# B&R Automation Studio project MotionTestBenchMaster (part 8)

#### SIKO_FB.st - Siko Manager
```iecst
(********************************************************************
 * COPYRIGHT - Sidel SpA
 ********************************************************************
 * Library: SIDEL
 * File: SIKO_FB.st
 * Author: 100383
 * Created: November 16, 2015
 ********************************************************************
 * Implementation of library SIDEL_CNTR
 ********************************************************************)

FUNCTION_BLOCK Siko_FB

	memset(ADR(Com),0,SIZEOF(Com));

	DeviceData.EmergencyOkFbk := IN_EmergencyOK;

	IF NOT IN_CommunicationOK THEN
		DeviceData.PositioningInProgress := FALSE;
		DeviceData.InPosition := FALSE;
		CounterRead := 0;
		CounterWrite := 0;
		DeviceData.CalibrationInProgress := FALSE;
		DeviceData.CommunicationFault := TRUE;
		RETURN;
	ELSE
		DeviceData.CommunicationFault := FALSE;
	END_IF

	IF CounterRead <> 0 OR CounterWrite <> 0 OR (DeviceData.CalibrationInProgress AND NOT DeviceData.Calibrate) THEN
		DeviceData.ReadOrWriteInProgress := TRUE;
	ELSE
		DeviceData.ReadOrWriteInProgress := FALSE;
	END_IF

	TReadAndWrite(IN:= DeviceData.ReadOrWriteInProgress, PT:= t#30s);
	DeviceData.ReadOrWriteError := TReadAndWrite.Q;

	IF DeviceData.ReadOrWriteError OR IN_Reset THEN
		CounterRead := 0;
		CounterWrite := 0;
		DeviceData.CalibrationInProgress := FALSE;
	END_IF

	Com.SIKO_FLR	:= IO.SIKO_FLR;
	Temp_HIW		:= IO.SIKO_FLR.HIW_L + (IO.SIKO_FLR.HIW_H * 16#10000);
	Temp_IN_PWE		:= IO.SIKO_FLR.PWE_L + (IO.SIKO_FLR.PWE_H * 16#10000);

	IF DeviceData.Data.SpindlePitch = 0 THEN
		KFactorReal := 1.0;
	ELSE
		KFactorReal := 100.0;
	END_IF

	DeviceData.CurrentPos := UDINT_TO_REAL(Temp_HIW) / KFactorReal;

	DeviceData.TargetOutsideSwLimit := (DeviceData.TargetPos > DeviceData.Data.UpperLimit) OR (DeviceData.TargetPos < DeviceData.Data.LowerLimit);

	IF EDGEPOS(DeviceData.StartPositioning AND IN_EmergencyOK AND NOT DeviceData.MotorDisabled AND NOT DeviceData.TargetOutsideSwLimit) THEN
		DeviceData.PositioningInProgress := TRUE;
	END_IF

	DeviceData.InPosition := ABS(DeviceData.TargetPos - DeviceData.CurrentPos) <= DeviceData.Data.PosWindows;

	SwitchOn := DeviceData.JogBackward OR DeviceData.JogForward OR DeviceData.PositioningInProgress;

	TPowerOn(IN:= SwitchOn, PT:= t#20s);

	Com.FLR_SIKO.STW.0 := IN_EmergencyOK AND TPowerOn.Q AND DeviceData.Enable AND NOT DeviceData.OnError;
	Com.FLR_SIKO.STW.1 := IN_EmergencyOK AND TPowerOn.Q AND DeviceData.Enable AND NOT DeviceData.OnError;

	Com.FLR_SIKO.STW.7 := IN_Reset;

	Com.FLR_SIKO.STW.5 := Com.SIKO_FLR.ZSW.2 AND NOT DeviceData.AbortPositioning;
	Com.FLR_SIKO.STW.4 := Com.SIKO_FLR.ZSW.2 AND NOT DeviceData.AbortPositioning;

	Com.FLR_SIKO.STW.3 := Com.SIKO_FLR.ZSW.4;

	IF DeviceData.Enable THEN
		DeviceData.MotorDisabled := FALSE;
	ELSIF NOT DeviceData.Enable AND NOT Com.SIKO_FLR.ZSW.4 THEN
		DeviceData.MotorDisabled := TRUE;
	END_IF

	DeviceData.OnError := Com.SIKO_FLR.ZSW.3;

	DeviceData.Warning := Com.SIKO_FLR.ZSW.8 AND Com.SIKO_FLR.ZSW.7;

	DeviceData.DeviceOutsideSwLimit := Com.SIKO_FLR.ZSW.14 OR (DeviceData.CurrentPos > DeviceData.Data.UpperLimit) OR (DeviceData.CurrentPos < DeviceData.Data.LowerLimit);

	Com.FLR_SIKO.STW.9 := Com.SIKO_FLR.ZSW.2 AND NOT DeviceData.OnError AND NOT DeviceData.PositioningInProgress AND	(DeviceData.JogForward XOR DeviceData.JogBackward);

	Com.FLR_SIKO.STW.15 := Com.FLR_SIKO.STW.9 AND DeviceData.JogBackward;

	Com.FLR_SIKO.STW.6 := DeviceData.PositioningInProgress AND NOT DeviceData.OnError AND Com.SIKO_FLR.ZSW.15 AND Com.SIKO_FLR.ZSW.13;

	IF Com.FLR_SIKO.STW.6 THEN
		Temp_HSW := REAL_TO_UDINT(DeviceData.TargetPos * KFactorReal);
	END_IF

	PositionFinished := ABS(DeviceData.TargetPos - DeviceData.CurrentPos) <= DeviceData.Data.PosWindows;

	IF DeviceData.TargetOutsideSwLimit OR DeviceData.OnError OR NOT IN_EmergencyOK OR DeviceData.MotorDisabled OR
	(DeviceData.InPosition AND Com.SIKO_FLR.ZSW.13) OR
	(PositionFinished AND Com.SIKO_FLR.ZSW.13) OR
	EDGEPOS(DeviceData.AbortPositioning) THEN
		DeviceData.PositioningInProgress := FALSE;
	END_IF

	RisingFrontRead := EDGEPOS((DeviceData.StartRead AND NOT DeviceData.ReadOrWriteInProgress) OR ReloadData);

	Com.FLR_SIKO.PKE := 0;

	IF NOT DeviceData.ReadOrWriteError THEN
		IF RisingFrontRead THEN
			CounterRead := 1;
			ReloadData := FALSE;
		END_IF

		CASE CounterRead OF
			1:	// Operative Mode
				Com.FLR_SIKO.PKE := 16#13A2;

				IF Com.SIKO_FLR.PKE = 16#13A2 THEN
					DeviceData.Data.OperationMode := UDINT_TO_INT(Temp_IN_PWE);
					CounterRead := CounterRead  + 1;
				END_IF

			2:	// Error Buffer [0]
				Com.FLR_SIKO.IND := 0;
				Com.FLR_SIKO.PKE := 16#63B1;

				IF Com.SIKO_FLR.PKE = 16#43B1 THEN
					IF Com.SIKO_FLR.IND = 0 THEN
						DeviceData.Data.FaultBuffer0 := UDINT_TO_INT(Temp_IN_PWE);
						CounterRead := CounterRead  + 1;
					END_IF
				END_IF

			3:	// Error Buffer [1]
				Com.FLR_SIKO.IND := 1;
				Com.FLR_SIKO.PKE := 16#63B1;

				IF Com.SIKO_FLR.PKE = 16#43B1 THEN
					IF Com.SIKO_FLR.IND = 1 THEN
						DeviceData.Data.FaultBuffer1 := UDINT_TO_INT(Temp_IN_PWE);
						CounterRead := CounterRead  + 1;
					END_IF
				END_IF

			4:	// Error Buffer [2]
				Com.FLR_SIKO.IND := 2;
				Com.FLR_SIKO.PKE := 16#63B1;

				IF Com.SIKO_FLR.PKE = 16#43B1 THEN
					IF Com.SIKO_FLR.IND = 2 THEN
						DeviceData.Data.FaultBuffer2 := UDINT_TO_INT(Temp_IN_PWE);
						CounterRead := CounterRead  + 1;
					END_IF
				END_IF

			5:	// Error Buffer [3]
				Com.FLR_SIKO.IND := 3;
				Com.FLR_SIKO.PKE := 16#63B1;

				IF Com.SIKO_FLR.PKE = 16#43B1 THEN
					IF Com.SIKO_FLR.IND = 3 THEN
						DeviceData.Data.FaultBuffer3 := UDINT_TO_INT(Temp_IN_PWE);
						CounterRead := CounterRead  + 1;
					END_IF
				END_IF

			6:	// Error Buffer [4]
				Com.FLR_SIKO.IND := 4;
				Com.FLR_SIKO.PKE := 16#63B1;

				IF Com.SIKO_FLR.PKE = 16#43B1 THEN
					IF Com.SIKO_FLR.IND = 4 THEN
						DeviceData.Data.FaultBuffer4 := UDINT_TO_INT(Temp_IN_PWE);
						CounterRead := CounterRead  + 1;
					END_IF
				END_IF

			7:	// Error Buffer [5]
				Com.FLR_SIKO.IND := 5;
				Com.FLR_SIKO.PKE := 16#63B1;

				IF Com.SIKO_FLR.PKE = 16#43B1 THEN
					IF Com.SIKO_FLR.IND = 5 THEN
						DeviceData.Data.FaultBuffer5 := UDINT_TO_INT(Temp_IN_PWE);
						CounterRead := CounterRead  + 1;
					END_IF
				END_IF

			8:	// Error Buffer [6]
				Com.FLR_SIKO.IND := 6;
				Com.FLR_SIKO.PKE := 16#63B1;

				IF Com.SIKO_FLR.PKE = 16#43B1 THEN
					IF Com.SIKO_FLR.IND = 6 THEN
						DeviceData.Data.FaultBuffer6 := UDINT_TO_INT(Temp_IN_PWE);
						CounterRead := CounterRead  + 1;
					END_IF
				END_IF

			9:	// Error Buffer [7]
				Com.FLR_SIKO.IND := 7;
				Com.FLR_SIKO.PKE := 16#63B1;

				IF Com.SIKO_FLR.PKE = 16#43B1 THEN
					IF Com.SIKO_FLR.IND = 7 THEN
						DeviceData.Data.FaultBuffer7 := UDINT_TO_INT(Temp_IN_PWE);
						CounterRead := CounterRead  + 1;
					END_IF
				END_IF

			10:	// Error Buffer [8]
				Com.FLR_SIKO.IND := 8;
				Com.FLR_SIKO.PKE := 16#63B1;

				IF Com.SIKO_FLR.PKE = 16#43B1 THEN
					IF Com.SIKO_FLR.IND = 8 THEN
						DeviceData.Data.FaultBuffer8 := UDINT_TO_INT(Temp_IN_PWE);
						CounterRead := CounterRead  + 1;
					END_IF
				END_IF

			11:	// Error Buffer [9]
				Com.FLR_SIKO.IND := 9;
				Com.FLR_SIKO.PKE := 16#63B1;

				IF Com.SIKO_FLR.PKE = 16#43B1 THEN
					IF Com.SIKO_FLR.IND = 9 THEN
						DeviceData.Data.FaultBuffer9 := UDINT_TO_INT(Temp_IN_PWE);
						CounterRead := CounterRead  + 1;
					END_IF
				END_IF

			12:	// P Gain
				Com.FLR_SIKO.PKE := 16#13E8;

				IF Com.SIKO_FLR.PKE = 16#13E8 THEN
					DeviceData.Data.PGain := UDINT_TO_INT(Temp_IN_PWE);
					CounterRead := CounterRead  + 1;
				END_IF

			13:	// I Gain
				Com.FLR_SIKO.PKE := 16#13E9;

				IF Com.SIKO_FLR.PKE = 16#13E9 THEN
					DeviceData.Data.IGain := UDINT_TO_INT(Temp_IN_PWE);
					CounterRead := CounterRead  + 1;
				END_IF

			14:	// D Gain
				Com.FLR_SIKO.PKE := 16#13EA;

				IF Com.SIKO_FLR.PKE = 16#13EA THEN
					DeviceData.Data.DGain := UDINT_TO_INT(Temp_IN_PWE);
					CounterRead := CounterRead  + 1;
				END_IF

			15:	// A Pos
				Com.FLR_SIKO.PKE := 16#13EB;

				IF Com.SIKO_FLR.PKE = 16#13EB THEN
					DeviceData.Data.APos := UDINT_TO_INT(Temp_IN_PWE);
					CounterRead := CounterRead  + 1;
				END_IF

			16:	// V Pos
				Com.FLR_SIKO.PKE := 16#13EC;

				IF Com.SIKO_FLR.PKE = 16#13EC THEN
					DeviceData.Data.VPos := UDINT_TO_INT(Temp_IN_PWE);
					CounterRead := CounterRead  + 1;
				END_IF

			17:	// V Jog
				Com.FLR_SIKO.PKE := 16#13F0;

				IF Com.SIKO_FLR.PKE = 16#13F0 THEN
					DeviceData.Data.VJog := UDINT_TO_INT(Temp_IN_PWE);
					CounterRead := CounterRead  + 1;
				END_IF

			18:	// SpindlePitch
				Com.FLR_SIKO.PKE := 16#13F4;

				IF Com.SIKO_FLR.PKE = 16#13F4 THEN
					DeviceData.Data.SpindlePitch := UDINT_TO_INT(Temp_IN_PWE) / 100;
					CounterRead := CounterRead  + 1;
				END_IF

			19:	// GearIn
				Com.FLR_SIKO.PKE := 16#13F2;

				IF Com.SIKO_FLR.PKE = 16#13F2 THEN
					DeviceData.Data.GearIn := UDINT_TO_INT(Temp_IN_PWE);
					CounterRead := CounterRead  + 1;
				END_IF

			20:	// GearOut
				Com.FLR_SIKO.PKE := 16#13F3;

				IF Com.SIKO_FLR.PKE = 16#13F3 THEN
					DeviceData.Data.GearOut := UDINT_TO_INT(Temp_IN_PWE);
					CounterRead := CounterRead  + 1;
				END_IF

			21:	// Toll Pos
				Com.FLR_SIKO.PKE := 16#13F1;

				IF Com.SIKO_FLR.PKE = 16#13F1 THEN
					DeviceData.Data.PosWindows := UDINT_TO_REAL(Temp_IN_PWE) / KFactorReal;
					CounterRead := CounterRead  + 1;
				END_IF

			22:	// Rotation
				Com.FLR_SIKO.PKE := 16#13F5;

				IF Com.SIKO_FLR.PKE = 16#13F5 THEN
					DeviceData.Data.SenseOfRotation := UDINT_TO_INT(Temp_IN_PWE);
					CounterRead := CounterRead  + 1;
				END_IF

			23:	// Upper limit
				Com.FLR_SIKO.PKE := 16#13F8;

				IF Com.SIKO_FLR.PKE = 16#13F8 OR Com.SIKO_FLR.PKE = 16#23F8 THEN
					DeviceData.Data.UpperLimit := UDINT_TO_REAL(Temp_IN_PWE) / KFactorReal;
					CounterRead := CounterRead  + 1;
				END_IF

			24:	// Lower limit
				Com.FLR_SIKO.PKE := 16#13F9;

				IF Com.SIKO_FLR.PKE = 16#13F9 OR Com.SIKO_FLR.PKE = 16#23F9 THEN
					DeviceData.Data.LowerLimit := UDINT_TO_REAL(Temp_IN_PWE) / KFactorReal;
					CounterRead := CounterRead  + 1;
				END_IF

			25:	// Calibration value
				Com.FLR_SIKO.PKE := 16#13FA;

				IF Com.SIKO_FLR.PKE = 16#13FA OR Com.SIKO_FLR.PKE = 16#23FA THEN
					DeviceData.Data.CalibrationValue := UDINT_TO_REAL(Temp_IN_PWE) / KFactorReal;
					CounterRead := CounterRead  + 1;
				END_IF

			26:	// Status word
				Com.FLR_SIKO.PKE := 16#13FC;

				IF Com.SIKO_FLR.PKE = 16#13FC THEN
					DeviceData.Data.SystemStatusWord := UDINT_TO_INT(Temp_IN_PWE);
					CounterRead := 0;
				END_IF

		END_CASE
	END_IF

	DeviceData.WriteEnabled := (DeviceData.MotorDisabled OR NOT DeviceData.PositioningInProgress) AND NOT DeviceData.ReadOrWriteInProgress AND NOT DeviceData.ReadOrWriteError AND NOT DeviceData.IllegalOperation;

	RisingFrontWrite := EDGEPOS(DeviceData.StartWrite);

	IF RisingFrontWrite AND DeviceData.WriteEnabled AND NOT DeviceData.ReadOrWriteError THEN
		DeviceData.Data.TimeoutPositioning	:= IN_TimeOutPositioning;
		DeviceData.Data.PosWindows			:= IN_PosWindows;
		DeviceData.Data.UpperLimit			:= IN_UpperLimit;
		DeviceData.Data.LowerLimit			:= IN_LowerLimit;
		DeviceData.Data.CalibrationValue	:= IN_CalibrationValue;

		DeviceData.Data.PGain			:= REAL_TO_INT(IN_PGain);
		DeviceData.Data.IGain			:= REAL_TO_INT(IN_IGain);
		DeviceData.Data.DGain			:= REAL_TO_INT(IN_DGain);
		DeviceData.Data.VPos			:= REAL_TO_INT(IN_VPos);
		DeviceData.Data.APos			:= REAL_TO_INT(IN_APos);
		DeviceData.Data.VJog			:= REAL_TO_INT(IN_VJog);
		DeviceData.Data.GearIn			:= REAL_TO_INT(IN_GearIn);
		DeviceData.Data.GearOut			:= REAL_TO_INT(IN_GearOut);
		DeviceData.Data.SpindlePitch	:= REAL_TO_INT(IN_SpindlePitch);
		DeviceData.Data.SenseOfRotation	:= REAL_TO_INT(IN_SenseOfRotation);
	END_IF

	IF NOT DeviceData.ReadOrWriteError THEN
		IF RisingFrontWrite THEN
			CounterWrite := 1;
		END_IF

		CASE CounterWrite OF
			1:	// Op Mode
				Com.FLR_SIKO.PKE := 16#23A2;
				Temp_OUT_PWE := 2;

				IF Com.SIKO_FLR.PKE = 16#13A2 THEN
					CounterWrite := CounterWrite + 1;
				END_IF

			2:	// Proportional Gain
				Com.FLR_SIKO.PKE := 16#23E8;
				Temp_OUT_PWE := DeviceData.Data.PGain;

				IF Com.SIKO_FLR.PKE = 16#13E8 THEN
					CounterWrite := CounterWrite + 1;
				END_IF

			3:	// Integral Gain
				Com.FLR_SIKO.PKE := 16#23E9;
				Temp_OUT_PWE := DeviceData.Data.IGain;

				IF Com.SIKO_FLR.PKE = 16#13E9 THEN
					CounterWrite := CounterWrite + 1;
				END_IF

			4:	// Derivative Gain
				Com.FLR_SIKO.PKE := 16#23EA;
				Temp_OUT_PWE := DeviceData.Data.DGain;

				IF Com.SIKO_FLR.PKE = 16#13EA THEN
					CounterWrite := CounterWrite + 1;
				END_IF

			5:	// Acc Positioning
				Com.FLR_SIKO.PKE := 16#23EB;
				Temp_OUT_PWE := DeviceData.Data.APos;

				IF Com.SIKO_FLR.PKE = 16#13EB THEN
					CounterWrite := CounterWrite + 1;
				END_IF

			6:	// Speed Positioning
				Com.FLR_SIKO.PKE := 16#23EC;
				Temp_OUT_PWE := DeviceData.Data.VPos;

				IF Com.SIKO_FLR.PKE = 16#13EC THEN
					CounterWrite := CounterWrite + 1;
				END_IF

			7:	// Speed Jog
				Com.FLR_SIKO.PKE := 16#23F0;
				Temp_OUT_PWE := DeviceData.Data.VJog;

				IF Com.SIKO_FLR.PKE = 16#13F0 THEN
					CounterWrite := CounterWrite + 1;
				END_IF

			8:	// GearIn
				Com.FLR_SIKO.PKE := 16#23F2;
				Temp_OUT_PWE := DeviceData.Data.GearIn;

				IF Com.SIKO_FLR.PKE = 16#13F2 THEN
					CounterWrite := CounterWrite + 1;
				END_IF

			9:	// GearOut
				Com.FLR_SIKO.PKE := 16#23F3;
				Temp_OUT_PWE := DeviceData.Data.GearOut;

				IF Com.SIKO_FLR.PKE = 16#13F3 THEN
					CounterWrite := CounterWrite + 1;
				END_IF

			10:	// SpinlePitch
				Com.FLR_SIKO.PKE := 16#23F4;
				Temp_OUT_PWE := DeviceData.Data.SpindlePitch * 100 ;

				IF Com.SIKO_FLR.PKE = 16#13F4 THEN
					CounterWrite := CounterWrite + 1;
				END_IF

			11:	// Position Windows
				Com.FLR_SIKO.PKE := 16#23F1;
				Temp_OUT_PWE := REAL_TO_INT(DeviceData.Data.PosWindows * KFactorReal);

				IF Com.SIKO_FLR.PKE = 16#13F1 THEN
					CounterWrite := CounterWrite + 1;
				END_IF

			12:	// Rotatation
				Com.FLR_SIKO.PKE := 16#23F5;
				Temp_OUT_PWE := DeviceData.Data.SenseOfRotation;

				IF Com.SIKO_FLR.PKE = 16#13F5 THEN
					CounterWrite := CounterWrite + 1;
				END_IF

			13:	// Upper Limit
				Com.FLR_SIKO.PKE := 16#33F8;
				Temp_OUT_PWE := REAL_TO_UDINT(DeviceData.Data.UpperLimit * KFactorReal);

				IF Com.SIKO_FLR.PKE = 16#23F8 THEN
					CounterWrite := CounterWrite + 1;
				ELSIF Com.SIKO_FLR.PKE = 16#73F8 THEN
					CounterWrite := CounterWrite + 2;
				END_IF

			14:	// Lower Limit
				Com.FLR_SIKO.PKE := 16#33F9;
				Temp_OUT_PWE := REAL_TO_UDINT(DeviceData.Data.LowerLimit * KFactorReal);

				IF Com.SIKO_FLR.PKE = 16#23F9 THEN
					CounterWrite := 50;
				END_IF

			15:	//Upper Limit error - Write Lower Limit
				Com.FLR_SIKO.PKE := 16#33F9;
				Temp_OUT_PWE := REAL_TO_UDINT(DeviceData.Data.LowerLimit * KFactorReal);

				IF Com.SIKO_FLR.PKE = 16#23F9 THEN
					CounterWrite := CounterWrite + 1;
				END_IF

			16: //Upper Limit error - Reweite Upper limit
				Com.FLR_SIKO.PKE := 16#33F8;
				Temp_OUT_PWE := REAL_TO_UDINT(DeviceData.Data.UpperLimit * KFactorReal);

				IF Com.SIKO_FLR.PKE = 16#23F8 THEN
					CounterWrite	:= 50;
				END_IF

			50: //Reset PWE
				Temp_OUT_PWE	:= 0;
				CounterWrite	:= 0;
				ReloadData := TRUE;
		END_CASE
	END_IF

	IF EDGEPOS(DeviceData.Calibrate AND DeviceData.WriteEnabled) THEN
		CounterCalibration := 1;
	END_IF

	CASE CounterCalibration OF
		1:
			DeviceData.Data.CalibrationValue := IN_CalibrationValue;
			DeviceData.CalibrationDone := FALSE;
			CounterCalibration := CounterCalibration + 1;

		2://Write Calibration Data
			Com.FLR_SIKO.PKE := 16#33FA;
			Temp_OUT_PWE := REAL_TO_UDINT(DeviceData.Data.CalibrationValue * KFactorReal);
			DeviceData.CalibrationInProgress := TRUE;

			IF Com.SIKO_FLR.PKE = 16#23FA THEN
				CounterCalibration := CounterCalibration + 1;
			END_IF

		3://Check Calibration Data
			IF ABS(Temp_IN_PWE - Temp_HIW) < 5 THEN
				DeviceData.CalibrationDone := TRUE;
				DeviceData.CalibrationInProgress := FALSE;
				CounterCalibration := 0;
			END_IF
	END_CASE

	IF ((DeviceData.Calibrate AND NOT DeviceData.CalibrationInProgress) OR RisingFrontWrite) AND NOT DeviceData.WriteEnabled THEN
		DeviceData.IllegalOperation := TRUE;
	ELSIF DeviceData.IllegalOperation AND IN_Reset THEN
		DeviceData.IllegalOperation := FALSE;
	END_IF

	IO.FLR_SIKO := Com.FLR_SIKO;
	IO.FLR_SIKO.PWE_H := UDINT_TO_UINT(SHR(Temp_OUT_PWE, 16));
	IO.FLR_SIKO.PWE_L := UDINT_TO_UINT(Temp_OUT_PWE AND 16#FFFF);
	IO.FLR_SIKO.HSW_H := UDINT_TO_UINT(SHR(Temp_HSW, 16));
	IO.FLR_SIKO.HSW_L := UDINT_TO_UINT(Temp_HSW AND 16#FFFF) ;

END_FUNCTION_BLOCK
```

#### PID_FF_Mod.st - FF calculation
```iecst
FUNCTION_BLOCK PID_FF_Mod
	IF SP1_ON THEN
		FF_SP2_Save := IN_FF_SP2;
		IF FF_SP2_Save >= IN_FF_SP1 THEN
			FF_SP2_Save := IN_FF_SP1;
		END_IF
		FF_SP2_Time.PT := REAL_TO_TIME(IN_SP1_SP2_Time/1000);
	END_IF

	FF_SP2_Time.IN := SP1_ON;
	FF_SP2_Time();

	IF NOT IN_Reset AND IN_Enable THEN
		IF ( IN_Raise_Step_Counter >= IN_Raise_Step ) OR ( IN_Raise_Step_Counter >= 100 ) THEN
			Running := TRUE;
			Lower_Ramp := TRUE;
		END_IF
	END_IF

	IF (NOT IN_Enable AND (( IN_Lower_Step_Counter >= IN_Lower_Step ) OR ( IN_Lower_Step_Counter >= 100 )))
		OR IN_Reset THEN
		Running := FALSE;
		SP1_ON := FALSE;
		SP2_ON := FALSE;
	END_IF

	FF_SP1_Recipe := (IN_FF_SP1);
	FF_SP2_Recipe := (IN_FF_SP2);
	Speed := IN_Actual_Speed;
	Max_Speed := MAX(IN_Size_Speed, 1);

	FF_SP1_Val := FF_SP1_Recipe * Speed;
	FF_SP1_Val := FF_SP1_Val / Max_Speed;

	FF_SP2_Val := FF_SP2_Recipe * Speed;
	FF_SP2_Val := FF_SP2_Val / Max_Speed;

	IF NOT Running AND NOT Lower_Ramp THEN
		FF_value_Out := 0.0;
	ELSIF NOT Running THEN
		Ramp_Time := 200.0;
		Ramp_Speed_R := (IN_Ramp_Speed);
		Ramp_Value := Ramp_Value - ((Ramp_Time /1000.0) * Ramp_Speed_R );
		IF Ramp_Value <= 0 THEN
			Lower_Ramp := FALSE;
			Ramp_Value := 0;
		END_IF
		FF_value_Out := Ramp_Value;
	ELSIF SP2_ON THEN
		FF_value_Out := FF_SP2_Val;
		Ramp_Value := FF_SP2_Val;
	ELSIF FF_SP2_Time.Q THEN
		Ramp_Time := 200.0;
		Ramp_Speed_R := (IN_Ramp_Speed);
		Ramp_Value := Ramp_Value - ((Ramp_Time /1000.0) * Ramp_Speed_R );
		IF Ramp_Value <= FF_SP2_Val THEN
			SP2_ON := TRUE;
			Ramp_Value := FF_SP2_Val;
		END_IF
		FF_value_Out := Ramp_Value;
	ELSIF SP1_ON THEN
		FF_value_Out := FF_SP1_Val;
		Ramp_Value := FF_SP1_Val;
	ELSE
		Ramp_Time := 200.0;
		Ramp_Speed_R := (IN_Ramp_Speed);
		Ramp_Value := Ramp_Value + ((Ramp_Time /1000.0) * Ramp_Speed_R );
		FF_value_Out := Ramp_Value;
		IF Ramp_Value >= FF_SP1_Val THEN
			SP1_ON := TRUE;
		END_IF
	END_IF

	OUT_FF_Value := FF_value_Out;
	OUT_FF_Value_Int := REAL_TO_INT(FF_value_Out);
END_FUNCTION_BLOCK
```

#### PID_FF_Pump.st - FF calculation
```iecst
FUNCTION_BLOCK PID_FF_Pump
//Pressure Head = (Frequency * Frequency * Kf ) - (Kpc * Flow * Flow)
//To find Kf:
//1. Container Block
//2. Filler Empty with Filling Valves Closed
//3. Search for right Kf until FF = PID Out

//To Find Kpc:
//1. Filler at Max Speed
//2. Filler full of containers, filling containers
//3. Search for right Kpc until FF = PID Out

//                   /^^^^^^^^^^^^^^^^^^^^^^^^^^^^^^^^^^^^^^^^^^^^
//Pump Frquency =  \/ ((Pressure Head) + Kpc * (Flow * Flow)) / Kf

//Pump Frequency [Hz]
//Pressure Head [mbar] --> mm
//Flow [m3/h]

IF NOT IN_Enable OR IN_Reset THEN
	OUT_FF	:= 0.0;
	RETURN;
END_IF

//Calculation of centrifugal force
//F_{cf}= m {\omega^2}{r} --> Omega is the Angular Velocity.
//Filler Angular Velocity
Omega := ((IN_Actual_Speed / IN_FV_Number) / (3600.0)) * 2.0 * 3.1415;

//Filler Radius
IF IN_Control_Type THEN //0=Control on Ring;1=Control on Product Pipe
	Radius := (IN_RingDiameter_mm / 2.0 / 1000.0);
ELSE
	Radius := 0.0;
END_IF

//Centrifugal Force [N], With Gravity Aceleration
IF IN_Control_Type THEN //0=Control on Ring;1=Control on Product Pipe
	CentrifugalForce := ((0.5 * Omega * Omega * Radius * Radius) / 9.81) * 1000.0;
ELSE
	CentrifugalForce := (((0.5 * Omega * Omega * Radius * Radius) / 9.81) * 1000.0)/100; //Convertion to mm of Product Pump In Ring Configuration
END_IF

IF IN_Control_Type THEN //0=Control on Ring;1=Control on Product Pipe
	Level_SP_Calculated := IN_Actual_SPmm + IN_PTF_FromFloor + IN_PTF_FromFV - CentrifugalForce;	//[mm] Of Water From The Floor To The SP Product Pump
ELSE
	Level_SP_Calculated := (IN_Actual_SPbar * 10197)- CentrifugalForce; // in test((IN_Actual_SPbar*1000) + IN_FV_FromFloor + 430 (*offset between fv and PTF on ring*)) - CentrifugalForce;	//[mm] Of Water From The Floor To The SP Product Pump In Ring Configuration
END_IF

IF IN_Control_Type THEN //0=Control on Ring;1=Control on Product Pipe
	PV_Product_Pump:= (IN_Actual_PVmm + IN_PTF_FromFloor + IN_PTF_FromFV) - IN_TankLevel_mm; //[mm] Of Water From The Floor on The PV Product Pump -Used For Pump Autotuning
ELSE
	PV_Product_Pump:= ((IN_Actual_PVbar * 1000)+ IN_FV_FromFloor + 430) - IN_TankLevel_mm; //[mm] Of Water From The Floor on The PV Product Pump In Ring Configuration
END_IF

//Hz For Actual Flowrate
Kpc_FlowRate_Filling := IN_Pump_Kpc * EXPT(((IN_FMCActualFlowrate/ 10.0) * 60.0) / 1000.0 , 2); //FF Calc on Filling Valves OPENED From FMC

//Real Set Point
Real_Level := Level_SP_Calculated - IN_TankLevel_mm;

//Calculated PV
IF IN_Control_Type THEN //0=Control on Ring;1=Control on Product Pipe
	Pid_PV_Calculated := (IN_Actual_PVmm + CentrifugalForce - IN_PTF_FromFV);
ELSE
	Pid_PV_Calculated := IN_Actual_PVbar;
END_IF

IF Pid_PV_Calculated > 0 THEN
	OUT_PID_PV := Pid_PV_Calculated;
ELSE
	OUT_PID_PV := 0.0;
END_IF

IF Pid_PV_Calculated > 0 THEN
	IF IN_Control_Type THEN //0=Control on Ring;1=Control on Product Pipe
		OUT_PID_SP := IN_Actual_SPmm + IN_PTF_FromFV - CentrifugalForce;
	ELSE
		OUT_PID_SP := IN_Actual_SPbar (*- (CentrifugalForce/1000)*);
	END_IF
ELSE
	OUT_PID_SP := 0.0;
END_IF

//Feed Forward Value for PID Control
IF SQRT((Kpc_FlowRate_Filling + Real_Level) / IN_Pump_Kf) >0 THEN
	OUT_FF := LIMIT(0,SQRT((Kpc_FlowRate_Filling + Real_Level) / IN_Pump_Kf),IN_Pump_OutMax);
ELSE
	OUT_FF := 0.0;
END_IF

//Detecting Wrong Setting
IF IN_Control_Type THEN //0=Control on Ring;1=Control on Product Pipe
	OUT_Error := IN_RingDiameter_mm =0.0 OR IN_PTF_FromFloor=0.0 OR IN_PTF_FromFV=0.0 OR IN_Pump_Kf=0.0 OR IN_Pump_Kpc=0.0 OR IN_Pump_OutMax=0.0;
ELSE
	OUT_Error := IN_FV_FromFloor=0.0 OR IN_Pump_Kf=0.0 OR IN_Pump_Kpc=0.0 OR IN_Pump_OutMax=0.0;
END_IF

END_FUNCTION_BLOCK

FUNCTION_BLOCK PID_FF_PumpH
//Pressure Head = (Frequency * Frequency * Kf ) - (Kpc * Flow * Flow)
//To find Kf:
//1. Container Block
//2. Filler Empty with Filling Valves Closed
//3. Search for right Kf until FF = PID Out

//To Find Kpc:
//1. Filler at Max Speed
//2. Filler full of containers, filling containers
//3. Search for right Kpc until FF = PID Out

//                  /^^^^^^^^^^^^^^^^^^^^^^^^^^^^^^^^^^^^^^^^^^^^
//Pump Frquency =  \/ ((Pressure Head) + Kpc * (Flow * Flow)) / Kf

//Pump Frequency [Hz]
//Pressure Head [mbar] --> mm
//Flow [m3/h]

IF NOT IN_Enable OR IN_Reset THEN
	OUT_FF	:= 0.0;
	RETURN;
END_IF

//Calculation of centrifugal force
//F_{cf}= m {\omega^2}{r} --> Omega is the Angular Velocity.
//Filler Angular Velocity
Omega := ((IN_Actual_Speed / IN_FV_Number) / (3600.0)) * 2.0 * 3.1415;

//Filler Radius
IF IN_Control_Type THEN //0=Control on Ring;1=Control on Product Pipe
	Radius := (IN_RingDiameter_mm / 2.0 / 1000.0);
ELSE
	Radius := 0.0;
END_IF

//Centrifugal Force [N], With Gravity Aceleration
IF IN_Control_Type THEN //0=Control on Ring;1=Control on Product Pipe
	CentrifugalForce := ((0.5 * Omega * Omega * Radius * Radius) / 9.81) * 1000.0;
ELSE
	CentrifugalForce := (((0.5 * Omega * Omega * Radius * Radius) / 9.81) * 1000.0)/100; //Convertion to mm of Product Pump In Ring Configuration
END_IF

//MAX Filling Time
MAX_FillingTime := (1000.0 / (IN_Recipe_Speed /3600.0)) * IN_FMCStepExitCam;

//Actual Filling Time
IF IN_FMCAverFillingTime >= 0 THEN
	Calculated_FillingTime := IN_FMCAverFillingTime;
ELSE
	Calculated_FillingTime := IN_PumpMaxFillingTime;
END_IF

FillingTime := MIN(Calculated_FillingTime,MAX_FillingTime);

//MAX Containers Number Into Filling Zone (Used only to control the value from the FMC "ITC_FMC_Tot_FV_Actual_In_Filling")
MAX_ContainersNumber := ((IN_Recipe_Speed * FillingTime / 3600000.0) - IN_FMCStepStartFilling);

IF IN_Control_Type THEN //0=Control on Ring;1=Control on Product Pipe
	Level_SP_Calculated := IN_Actual_SPmm + IN_PTF_FromFloor + IN_PTF_FromFV - CentrifugalForce;	//[mm] Of Water From The Floor To The SP Product Pump
ELSE
	Level_SP_Calculated := ((IN_Actual_SPbar*1000)+ IN_FV_FromFloor + 430(*offset between fv and PTF on ring*)) - CentrifugalForce;	//[mm] Of Water From The Floor To The SP Product Pump In Ring Configuration
END_IF

IF IN_Control_Type THEN //0=Control on Ring;1=Control on Product Pipe
	PV_Product_Pump:= (IN_Actual_PVmm + IN_PTF_FromFloor + IN_PTF_FromFV) - IN_TankLevel_mm; //[mm] Of Water From The Floor on The PV Product Pump -Used For Pump Autotuning
ELSE
	PV_Product_Pump:= ((IN_Actual_PVbar *1000)+ IN_FV_FromFloor + 430) - IN_TankLevel_mm; //[mm] Of Water From The Floor on The PV Product Pump In Ring Configuration
END_IF

//Hz For Actual Flowrate
Kpc_FlowRate_Filling := IN_Pump_Kpc * EXPT(((IN_FMCActualFlowrate/ 10.0) * 60.0) / 1000.0 , 2); //FF Calc on Filling Valves OPENED From FMC

//Real Set Point
Real_Level := Level_SP_Calculated - IN_TankLevel_mm;

//Centrifugal Force
OUT_Centifrugal := CentrifugalForce;

//Feed Forward Value for PID Control
IF SQRT((Kpc_FlowRate_Filling + Real_Level) / IN_Pump_Kf) >0 THEN
	OUT_FF := LIMIT(0,SQRT((Kpc_FlowRate_Filling + Real_Level) / IN_Pump_Kf),IN_Pump_OutMax);
ELSE
	OUT_FF := 0.0;
END_IF

//Detecting Wrong Setting
IF IN_Control_Type THEN //0=Control on Ring;1=Control on Product Pipe
OUT_Error := IN_RingDiameter_mm =0.0 OR IN_PTF_FromFloor=0.0 OR IN_PTF_FromFV=0.0 OR
			 IN_Pump_Kf=0.0 OR IN_Pump_Kpc=0.0 OR IN_Pump_OutMax=0.0 OR IN_FMCAverFillingTime=0.0 OR
			 IN_FMCStepStartFilling= 0.0 OR IN_FMCStepExitCam=0.0;
ELSE
	OUT_Error := IN_FV_FromFloor=0.0 OR IN_Pump_Kf=0.0 OR IN_Pump_Kpc=0.0 OR IN_Pump_OutMax=0.0;
END_IF

END_FUNCTION_BLOCK
```

#### Sequencer.st
```iecst
FUNCTION_BLOCK Sequencer_v1
	VAR_ChangeInProgress := OUT_JMP_Step <> IN_Step;

	IF VAR_ChangeInProgress THEN
		memset(ADR(TON_Time),	0,	SIZEOF(TON_Time));
		memset(ADR(T_Time),		0,	SIZEOF(T_Time));
		memset(ADR(TO_Time),	0,	SIZEOF(TO_Time));
		OUT_JMP_StepPrevious := OUT_JMP_Step ;
	END_IF

	//Volatile Timer
	TON_Time(
	IN := IN_StepConfig.TON_TimeSTART AND NOT VAR_ChangeInProgress AND NOT IN_Pause_Request,
	PT := UINT_TO_TIME(IN_StepConfig.TON_TimePr * 1000)
	);
	OUT_TON_Time_END := TON_Time.Q;

	//Retentive Counter
	T_Time(
	CU 		:= IN_T_TimeClock AND IN_StepConfig.T_TimeSTART AND NOT IN_StepConfig.T_TimeSTOP AND NOT IN_Pause_Request,
	RESET 	:= IN_StepConfig.T_TimeRESET OR VAR_ChangeInProgress,
	PV 		:= IN_StepConfig.T_TimePr
	);
	OUT_T_Time_END := T_Time.Q;

	//Volatile Timeout
	TO_Time(
	IN := NOT VAR_ChangeInProgress,
	PT := UINT_TO_TIME(IN_StepConfig.TO_TimePr * 1000)
	);
	OUT_TO_Time_END := TO_Time.Q;

	//Reset counter Initialized to wait counter reset from Filler
	IF VAR_ChangeInProgress THEN
		VAR_CounterInitialized := FALSE;
	END_IF

	//Eneble Laps Counter Request only if the counter is initialized
	IF NOT VAR_CounterInitialized THEN
		OUT_LapsCounterRequest := FALSE;
	ELSIF IN_StepConfig.Laps_Counter_Enable THEN
		OUT_LapsCounterRequest := TRUE;
	END_IF

	//Step Counter is initialized when the value is 0
	IF IN_StepCounter = 0 THEN
		VAR_CounterInitialized := TRUE;
	END_IF

	//Laps Progress
	OUT_Laps_Progress := (IN_StepCounter / MAX(1, IN_FillingValveNr));

	//Laps Expired
	OUT_Laps_Done := OUT_Laps_Progress >= IN_StepConfig.Laps_Request AND IN_StepCounter > 0 AND IN_StepConfig.Laps_Counter_Enable;

	OUT_JMP_Step 	:= IN_Step;
	OUT_HMI_ID		:= IN_StepConfig.HMI_ID;

	//Cycles
	IF CyclesCounter >= IN_StepConfig.Cycle_Pr THEN
		OUT_Cycles_Done := TRUE;
	ELSE
		OUT_Cycles_Done:= FALSE;
	END_IF

	//Timers Visualization
	OUT_StepTimePr_TON  := REAL_TO_UINT(TIME_TO_REAL(TON_Time.PT) / 1000.0);
	OUT_StepTimePr_T    := T_Time.PV;
	OUT_StepTimeCV_TON	:= REAL_TO_UINT(TIME_TO_REAL(TON_Time.ET) / 1000.0);
	OUT_StepTimeCV_T    := T_Time.CV;

END_FUNCTION_BLOCK

FUNCTION_BLOCK Sequencer_v2
	VAR_ChangeInProgress := OUT_StepActual <> IN_Step; //v2

	IF VAR_ChangeInProgress THEN
		memset(ADR(TON_Time),	0,	SIZEOF(TON_Time));
		memset(ADR(T_Time),		0,	SIZEOF(T_Time));
		memset(ADR(TO_Time),	0,	SIZEOF(TO_Time));
		OUT_StepPrevious := OUT_StepActual; //v2
	END_IF

	//Volatile Timer
	TON_Time(
	IN := IN_StepConfig.TON_TimeSTART AND NOT VAR_ChangeInProgress AND NOT IN_Pause_Request,
	PT := UINT_TO_TIME(IN_StepConfig.TON_TimePr * 1000)
	);
	OUT_TON_Time_END := TON_Time.Q;

	//Retentive Counter
	T_Time(
	CU 		:= IN_T_TimeClock AND IN_StepConfig.T_TimeSTART AND NOT IN_StepConfig.T_TimeSTOP AND NOT IN_Pause_Request,
	RESET 	:= IN_StepConfig.T_TimeRESET OR VAR_ChangeInProgress,
	PV 		:= IN_StepConfig.T_TimePr
	);
	OUT_T_Time_END := T_Time.Q;

	//Volatile Timeout
	TO_Time(
	IN := NOT VAR_ChangeInProgress,
	PT := UINT_TO_TIME(IN_StepConfig.TO_TimePr * 1000)
	);
	OUT_TO_Time_END := TO_Time.Q;

	//Progressive Time v2
	T_StepProgressiveTime(
	IN := NOT VAR_ChangeInProgress,
	PT := T#24d,
	);

	//Reset counter Initialized to wait counter reset from Filler
	IF VAR_ChangeInProgress THEN
		VAR_CounterInitialized := FALSE;
	END_IF

	//Eneble Laps Counter Request only if the counter is initialized
	IF NOT VAR_CounterInitialized THEN
		OUT_LapsCounterRequest := FALSE;
	ELSIF IN_StepConfig.Laps_Counter_Enable THEN
		OUT_LapsCounterRequest := TRUE;
	END_IF

	//Step Counter is initialized when the value is 0
	IF IN_StepCounter = 0 THEN
		VAR_CounterInitialized := TRUE;
	END_IF

	//Laps Progress
	OUT_Laps_Progress := (IN_StepCounter / MAX(1, IN_FillingValveNr));

	//Laps Expired
	OUT_Laps_Done := OUT_Laps_Progress >= IN_StepConfig.Laps_Request AND IN_StepCounter > 0 AND IN_StepConfig.Laps_Counter_Enable;

	OUT_StepActual 	:= IN_Step; //v2
	OUT_HMI_ID		:= IN_StepConfig.HMI_ID;

	//Cycles
	IF CyclesCounter >= IN_StepConfig.Cycle_Pr THEN
		OUT_Cycles_Done := TRUE;
	ELSE
		OUT_Cycles_Done:= FALSE;
	END_IF

	//Timers Visualization
	OUT_StepTimePr_TON  	:= REAL_TO_UINT(TIME_TO_REAL(TON_Time.PT) / 1000.0);
	OUT_StepTimePr_T    	:= T_Time.PV;
	OUT_StepTimeCV_TON		:= REAL_TO_UINT(TIME_TO_REAL(TON_Time.ET) / 1000.0);
	OUT_StepTimeCV_T    	:= T_Time.CV;
	OUT_StepProgressiveTime	:= REAL_TO_UINT(TIME_TO_REAL(T_StepProgressiveTime.ET) / 1000.0); //v2

END_FUNCTION_BLOCK
```

#### TankLevel.st
```iecst
FUNCTION_BLOCK TankMultiScale
	IF IN_ProbeLength_mm = 0.0 OR IN_TNK_Diameter_mm = 0.0 THEN
		RETURN;
	END_IF

	//Index [0]: level in percentage
	//Index [1]: volume in liters
	//Index [2]: height in mm
	//Index [3]: HMI_PAR_2._309

	pi 			:= 3.14;
	diameter_cm	:= IN_TNK_Diameter_mm / 10.0; 	// [cm]
	r_cm  		:= diameter_cm / 2.0;			// [cm]

	heightTot_cm		:= IN_ProbeLength_mm / 10.0; 	// [cm]
	volumeTot_cm3 		:= (pi * r_cm * r_cm) * heightTot_cm;	// [cm3]
	volumeTot_liters 	:= volumeTot_cm3 / 1000;			// [dm3]/[l]

	heightAck_cm		:= IN_ProbeLength_mm / 10.0 * IN_TNK_PV / 100.0;	// [cm]
	volumeAck_cm3 		:= (pi * r_cm * r_cm) * heightAck_cm;	// [cm3]
	volumeAck_liters 	:= volumeAck_cm3 / 1000;			// [dm3]/[l]

	LowLimitAbs_cm		:= IN_ProbeLength_mm / 10.0 * IN_TNK_LowLimitAbs / 100.0;	// [cm]
	LowLimitAbs_cm3		:= (pi * r_cm * r_cm) * LowLimitAbs_cm;	// [cm3]
	LowLimitAbs_liters 	:= LowLimitAbs_cm3 / 1000;			// [dm3]/[l]

	OUT_Scale[0].ActValue	:=	LIMIT(IN_Scale[0].ScaleLOW, IN_TNK_PV, IN_Scale[0].ScaleHIGH);
	IF IN_TNK_PV > 1.0 THEN
		OUT_Scale[1].ActValue := volumeAck_liters + IN_TNK_Bottom_liters;
	ELSE
		OUT_Scale[1].ActValue := 0.0;
	END_IF

	OUT_Scale[2].ActValue 	:= (OUT_Scale[0].ActValue * IN_ProbeLength_mm / 100.0)(* + IN_FromFloor_ToZeroProbe_mm*);

	OUT_Scale[3].ActValue := LowLimitAbs_liters + IN_TNK_Bottom_liters;

	CASE IN_Sp_Type OF
		0:
			HMI.SP[0] 		:= IN_Scale[0].ActualSP;
			HMI.SP[1]		:= IN_Scale[1].ActualSP;
			HMI.SP[2]		:= IN_Scale[2].ActualSP;
			HMI.SP[3]		:= IN_Scale[3].ActualSP;
			HMI.Wait[0] 	:= FALSE;
			HMI.Wait[1]		:= FALSE;
			HMI.Wait[2]		:= FALSE;
			HMI.Wait[3]		:= FALSE;

		1:	// Wait percentage SP
			HMI.SP[0] 		:= IN_Scale[0].ActualSP;
			HMI.SP[1]		:= (IN_Scale[0].ActualSP * volumeTot_liters) / 100.0;
			HMI.SP[2]		:= (IN_Scale[0].ActualSP * IN_ProbeLength_mm / 100.0) + IN_FromFloor_ToZeroProbe_mm;
			HMI.SP[3]		:= IN_Scale[3].ActualSP;
			HMI.Wait[0] 	:= IN_Wait;
			HMI.Wait[1]		:= FALSE;
			HMI.Wait[2]		:= FALSE;
			HMI.Wait[3]		:= FALSE;

		2:	// Wait Volume SP
			HMI.SP[0]		:= ((IN_Scale[1].ActualSP - IN_TNK_Bottom_liters) / volumeTot_liters) *100.0;
			HMI.SP[1]		:= IN_Scale[1].ActualSP;
			HMI.SP[2]		:= (((IN_Scale[1].ActualSP / volumeTot_liters) *100.0) * IN_ProbeLength_mm /100.0) + IN_FromFloor_ToZeroProbe_mm;
			HMI.SP[3]		:= IN_Scale[3].ActualSP;
			HMI.Wait[0] 	:= FALSE;
			HMI.Wait[1]		:= IN_Wait;
			HMI.Wait[2]		:= FALSE;
			HMI.Wait[3]		:= FALSE;

		3:	// Wait level Height
			HMI.SP[0] 		:= (IN_Scale[2].ActualSP - IN_FromFloor_ToZeroProbe_mm) / IN_ProbeLength_mm  *100.0;
			HMI.SP[1]		:= (HMI.SP[0] * volumeTot_liters) / 100.0 + IN_TNK_Bottom_liters;
			HMI.SP[2]		:= IN_Scale[2].ActualSP;
			HMI.SP[3]		:= IN_Scale[3].ActualSP;
			HMI.Wait[0] 	:= FALSE;
			HMI.Wait[1]		:= FALSE;
			HMI.Wait[2]		:= IN_Wait;
			HMI.Wait[3]		:= FALSE;
	END_CASE

	HMI.ConfigPresent	:= IN_ConfigPresent;
	HMI.PV[0] 			:= OUT_Scale[0].ActValue;
	HMI.PV[1] 			:= OUT_Scale[1].ActValue;
	HMI.PV[2] 			:= OUT_Scale[2].ActValue;
	HMI.PV[3] 			:= OUT_Scale[3].ActValue;

END_FUNCTION_BLOCK
```

#### TP_Reset.st
```iecst
FUNCTION_BLOCK TP_Reset
	RT_Info(enable := TRUE);

	IF EDGEPOS(IN) THEN
		TimeCounter	:= TIME_TO_UDINT(PT) * 1000;	//micros
	END_IF

	IF TimeCounter >= RT_Info.cycle_time THEN
		TimeCounter := TimeCounter - (RT_Info.cycle_time);
	ELSE
		TimeCounter := 0;
	END_IF

	IF EDGEPOS(RESET) THEN
		TimeCounter := 0;
	END_IF

	Q := TimeCounter <> 0;
END_FUNCTION_BLOCK
```

#### FB_Flip.st
```iecst
FUNCTION_BLOCK FB_Flip
	TON_Blink.IN := NOT TON_Blink.Q;
	TON_Blink.PT := t#1s;
	TON_Blink();

	IF EDGEPOS(TON_Blink.Q) THEN
		VAR_CyleOn 		:= FALSE;
		VAR_CyleCntOn	:= FALSE;
		VAR_CyleCntOff	:= FALSE;
		VAR_CyleOnTimeReset := FALSE;
		VAR_CyleOffTimeReset:= FALSE;
		VAR_CyleNrReset	:= FALSE;
		VAR_CycleNrDone	:= FALSE;
		CASE Command_State OF
			0:
				IF IN_CycleOn AND NOT IN_CyclePause THEN
					IF IN_CycleStartOffCount THEN
						Command_State := 2;
					ELSIF IN_CycleTimeOn > 0 THEN
						Command_State := 1;
					END_IF
				END_IF

			1:	//ON TIME
				VAR_CyleOn 		:= TRUE;
				VAR_CyleCntOn	:= TRUE;
				VAR_CyleOffTimeReset	:= TRUE;

				IF NOT IN_CycleOn THEN
					Command_State := 99; // //RESET CNT
				ELSIF IN_CyclePause THEN
					Command_State := 10; // PAUSE CMD
				ELSE
					IF VAR_CycleOnDone THEN
						VAR_CyleOnTimeReset := TRUE;
						IF IN_CycleLoop THEN
							IF IN_CycleTimeOff > 0 THEN
								Command_State := 2; //PAUSE TIME
							END_IF
						ELSE
							VAR_CycleNr 	:= MIN(VAR_CycleNr  +1, IN_CycleNr);
							 IF (IN_CycleNr = VAR_CycleNr) AND NOT IN_CycleLoop THEN
								Command_State := 3; // DONE
							ELSE
								Command_State := 2; //PAUSE TIME
							END_IF
						END_IF
					END_IF
				END_IF

			2: //PAUSE TIME

				VAR_CyleCntOff	:= NOT IN_CyclePause;
				VAR_CyleOnTimeReset	:= TRUE;

				IF NOT IN_CycleOn THEN
					Command_State := 99; // //RESET CNT
				ELSIF VAR_CycleOffDone AND NOT IN_CyclePause THEN
					VAR_CyleOffTimeReset := TRUE;
					IF VAR_CycleNrDone THEN
						Command_State := 3; // DONE
					ELSIF IN_CycleTimeOn > 0 THEN
						Command_State := 1; // ON TIME
					END_IF
				END_IF

			3: // DONE
				VAR_CycleNrDone	:= TRUE;
				IF NOT IN_CycleOn OR IN_CycleLoop THEN
					Command_State := 99; // //RESET CNT
				END_IF

			10: // PAUSE

				IF NOT IN_CycleOn THEN
					Command_State := 99; // //RESET CNT
				ELSIF NOT IN_CyclePause THEN
					Command_State := 1; // OFF
				END_IF

			99: //RESET CNT
				VAR_CyleOnTimeReset := TRUE;
				VAR_CyleOffTimeReset:= TRUE;
				VAR_CycleNr := 0;
				Command_State := 0; // OFF
		END_CASE

		IF VAR_CyleCntOn THEN
			VAR_CycleTimeOn := MIN(VAR_CycleTimeOn  +1, IN_CycleTimeOn);
			VAR_CycleOnDone := IN_CycleTimeOn = VAR_CycleTimeOn;
		ELSE
			VAR_CycleOnDone := FALSE;
		END_IF

		IF VAR_CyleCntOff THEN
			VAR_CycleTimeOff := MIN(VAR_CycleTimeOff +1, IN_CycleTimeOff);
			VAR_CycleOffDone := IN_CycleTimeOff = VAR_CycleTimeOff;
		ELSE
			VAR_CycleOffDone := FALSE;
		END_IF

		IF VAR_CyleOffTimeReset THEN
			VAR_CycleTimeOff := 0;
		END_IF
		IF VAR_CyleOnTimeReset THEN
			VAR_CycleTimeOn := 0;
		END_IF
		IF IN_CycleNrReset THEN
			VAR_CycleNr 	:= 0;
		END_IF

		Out 			:= VAR_CyleOn;
		OUT_CycleNr		:= VAR_CycleNr;
		OUT_CycleTimeOn	:= VAR_CycleTimeOn;
		OUT_CycleTimeOff:= VAR_CycleTimeOff;
		OUT_CycleDone 	:= VAR_CycleNrDone;
	END_IF
END_FUNCTION_BLOCK
```

#### Constant.var
```iecst
(*ITC*)
VAR CONSTANT
	CST_MinITCPartner : USINT := 11;
	CST_MaxITCPartner : USINT := 89; (*V4.A.A.1.6.12*)
END_VAR
(*HMI Rele Station and Channel State*)
VAR CONSTANT
	CST_MAX_Nr_Channels : USINT := 16;
	CST_RELE_NO_COMMUN : USINT := 0; (*White + X Red Symbol*)
	CST_RELE_ON : USINT := 1; (*Green*)
	CST_RELE_ON_BY_PLC : USINT := 2; (*Green*)
	CST_RELE_ON_WARNING : USINT := 3; (*Green + Warning Symbol*)
	CST_RELE_ON_CONFIG_ERROR : USINT := 4; (*Green + Yellow with X Blue*)
	CST_RELE_OFF_FAULT : USINT := 5; (*Black + Fault Symbol*)
	CST_RELE_OFF_BY_PB_HW : USINT := 6; (*Black + HW Symbol*)
	CST_RELE_OFF_BY_HMI : USINT := 7; (*Black + HMI Symbol*)
	CST_RELE_OFF_BY_PLC : USINT := 8; (*Black + PLC Symbol*)
	CST_RELE_OFF : USINT := 9; (*Black*)
	CST_RELE_OFF_CONFIG_ERROR : USINT := 10; (*Black + Yellow with X Blue*)
	CST_RELE_NOT_DEFINE : USINT := 11; (*Yellow + X Blue*)
END_VAR
```

### Library Logical/00_AID/Libraries/Sidel_Libraries/Sidel_Obj (IEC)

#### Sidel_Obj.fun - Exported functions and function blocks
```iecst
FUNCTION_BLOCK Analog_In_Direct_Inverse
	VAR_INPUT
		IN_ConfigPresent : BOOL;
		IN_Simulation : BOOL;
		IN_0_20mA : BOOL;
		IN_FaultOutMode : USINT; (*LowOnFault(1) ; HighOnFault (2) HoldOnFault (0)*)
		IN_EngScale : BOOL;
		IN_CompareMode : USINT; (*0 = Off, 1 = PV_Greater_SP, 2 = PV_Less_SP, 3 = PV_Equal_SP, 4 = On*)
		IN_ScaleLOW : REAL;
		IN_ScaleHIGH : REAL;
		IN_AlarmEn : BOOL;
		IN_MaskEn : BOOL;
		IN_ConfigPopup : BOOL;
		IN_Reset : BOOL; (*Reset Analog Channel Alarm*)
		IN_ActualSP : REAL; (*Signal Input Actual Set Point*)
		IN_MinDev : REAL; (*To Set Point Low Deviation (for SP obtained)*)
		IN_MaxDev : REAL; (*To Set Point High Deviation (for SP obtained)*)
		IN_WaitDelay : TIME;
		IN_HighLimitEn : BOOL;
		IN_HighLimitSP : REAL;
		IN_HighLimitHyst : REAL;
		IN_HighLimitDelay : TIME;
		IN_LowLimitEn : BOOL;
		IN_LowLimitSP : REAL;
		IN_LowLimitHyst : REAL;
		IN_LowLimitDelay : TIME;
		IN_Direct_Inverse : BOOL; (*Read Mode: "0" for Direct "1" for Inverse*)
		IN_Delta : REAL; (*Delta Value for Real Component Height*)
	END_VAR
	VAR_OUTPUT
		OUT_ActValue : REAL; (*Manipulated value*)
		OUT_SpReached : BOOL; (*Output Set Point Reached*)
		OUT_HighLimit : BOOL;
		OUT_LowLimit : BOOL;
		OUT_Alarm : BOOL; (*Output Fault*)
		OUT_RawOverflow : BOOL; (*Output Fault*)
		OUT_RawUnderflow : BOOL; (*Output Fault*)
	END_VAR
	VAR_IN_OUT
		IO : IO_Analog_IN_Type;
		HMI : HMI_Analog_IN_Type;
	END_VAR
	VAR
		VAR_Fault : BOOL; (*Alarm Output for Fault or Warning*)
		VAR_Mask : BOOL;
		VAR_Out : REAL;
		VAR_ChannelActive : BOOL;
		VAR_Wait : BOOL;
		VAR_iFault : BOOL;
		VAR_SpReached : BOOL;
		LCRLimScal_0_20mA : LCRLimScal;
		LCRLimScal_4_20mA : LCRLimScal;
		TMR_TON_HighLimitDelay : TON;
		TMR_TON_LowLimitDelay : TON;
		TMR_TOF_SpReached : TOF;
	END_VAR
END_FUNCTION_BLOCK

FUNCTION_BLOCK Analog_In
	VAR_INPUT
		IN_ConfigPresent : BOOL;
		IN_Simulation : BOOL;
		IN_0_20mA : BOOL;
		IN_FaultOutMode : USINT; (*LowOnFault(1) ; HighOnFault (2) HoldOnFault (0)*)
		IN_EngScale : BOOL;
		IN_CompareMode : USINT; (*0 = Off, 1 = PV_Less_SP, 2 = PV_Greater_SP, 3 = PV_Equal_SP, 4 = Reached On*)
		IN_ScaleLOW : REAL;
		IN_ScaleHIGH : REAL;
		IN_AlarmEn : BOOL;
		IN_MaskEn : BOOL;
		IN_ConfigPopup : BOOL;
		IN_Reset : BOOL; (*Reset Analog Channel Alarm*)
		IN_ActualSP : REAL; (*Signal Input Actual Set Point*)
		IN_MinDev : REAL; (*To Set Point Low Deviation (for SP obtained)*)
		IN_MaxDev : REAL; (*To Set Point High Deviation (for SP obtained)*)
		IN_WaitDelay : TIME;
		IN_HighLimitEn : BOOL;
		IN_HighLimitSP : REAL;
		IN_HighLimitHyst : REAL;
		IN_HighLimitDelay : TIME;
		IN_LowLimitEn : BOOL;
		IN_LowLimitSP : REAL;
		IN_LowLimitHyst : REAL;
		IN_LowLimitDelay : TIME;
		IN_TotPulseWeight : REAL;
		IN_TotType : USINT;
		IN_PLCCounterEn : BOOL;
		IN_PLCCounterSP : REAL;
		IN_PLCCounterReset : BOOL;
		IN_HMITotEn : BOOL;
		IN_HMITotReset : BOOL;
	END_VAR
	VAR_OUTPUT
		OUT_ActValue : REAL; (*Manipulated value*)
		OUT_SpReached : BOOL; (*Output Set Point Reached*)
		OUT_HighLimit : BOOL;
		OUT_LowLimit : BOOL;
		OUT_Alarm : BOOL; (*Output Fault*)
		OUT_RawOverflow : BOOL; (*Output Fault*)
		OUT_RawUnderflow : BOOL; (*Output Fault*)
		OUT_PLCCounterReached : BOOL; (*Output Fault*)
	END_VAR
	VAR_IN_OUT
		IO : IO_Analog_IN_Type;
		HMI : HMI_Analog_IN_Type;
	END_VAR
	VAR
		VAR_Fault : BOOL; (*Alarm Output for Fault or Warning*)
		VAR_Mask : BOOL;
		VAR_Out : REAL;
		VAR_ChannelActive : BOOL;
		VAR_Wait : BOOL;
		VAR_iFault : BOOL;
		VAR_SpReached : BOOL;
		LCRLimScal_0_20mA : LCRLimScal;
		LCRLimScal_4_20mA : LCRLimScal;
		HMITotalizer : AnalogTotalizer;
		PLCCounter : AnalogTotalizer;
		TMR_TON_HighLimitDelay : TON;
		TMR_TON_LowLimitDelay : TON;
		TMR_TOF_SpReached : TOF;
		TON_ChannelOk : TON;
	END_VAR
END_FUNCTION_BLOCK

FUNCTION_BLOCK GateDoorDigital_Obj
	VAR_INPUT
		IN_ConfigPresent : BOOL; (*Configuration: Device Present*)
		IN_Alarm : BOOL; (*Configuration: Timeout Alarm Control Enable*)
		IN_AlarmOpenReq : BOOL; (*Control: On State Time Out Alarm Request*)
		IN_AlarmCloseReq : BOOL; (*Control: Off State Time Out Alarm Request*)
		IN_SwitchDelay : TIME; (*Time: Row Input Switching State Display Delay*)
		IN_WaitOpen : BOOL; (*Control: On State Wait Request*)
		IN_WaitClose : BOOL; (*Control: Off State Wait Request*)
		IN_OnDelay : TIME; (*Time: State On / Alarm On Time Delay*)
		IN_OffDelay : TIME; (*Time: State Off / Alarm Off Time Delay*)
		IN_Reset : BOOL; (*Control: Alarm Reset Push Button*)
		IN_SafetyClosed : BOOL; (*From Safety: Gate Closed*)
		IN_SafetyShortCircuit : BOOL; (*From Safety: Short circuit or 1oo2*)
	END_VAR
	VAR_OUTPUT
		OUT_Opened : BOOL; (*OUT: Gate Opened*)
		OUT_Closed : BOOL; (*OUT: Gate Closed*)
		OUT_Alarm : BOOL; (*State On / Off Time Out Alarm*)
	END_VAR
	VAR_IN_OUT
		IO_Production : IO_Digital_IN_Type; (*State: Digital Input Structure*)
		HMI : HMI_GateDoor_Type;
	END_VAR
	VAR
		TMR_TON_ProdSwOn : TON;
		TMR_TON_ProdSwOff : TON;
		TMR_TON_CleanSwOn : TON;
		TMR_TON_CleanSwOff : TON;
		TMR_TON_ProdOnAlarm : TON;
		TMR_TON_ProdOffAlarm : TON;
		TMR_TON_CleanOnAlarm : TON;
		TMR_TON_CleanOffAlarm : TON;
		VAR_Signal : BOOL;
		VAR_ProdFault : BOOL;
		VAR_CleanFault : BOOL;
	END_VAR
END_FUNCTION_BLOCK

FUNCTION_BLOCK Analog_In_Multiscale
	VAR_INPUT
		IN_ConfigPresent : BOOL;
		IN_Simulation : BOOL;
		IN_0_20mA : BOOL;
		IN_MaskEn : BOOL;
		IN_Reset : BOOL; (*Reset Analog Channel Alarm*)
		IN_FaultOutMode : USINT; (*LowOnFault(1) ; HighOnFault (2) HoldOnFault (0)*)
		IN_EngScale : BOOL;
		IN_AlarmEn : BOOL;
		IN_ConfigPopup : BOOL;
		IN_PLCCounterEn : BOOL;
		IN_CompareMode : USINT; (*0 = Off, 1 = PV_Greater_SP, 2 = PV_Less_SP, 3 = PV_Equal_SP, 4 = On*)
		IN_ScaleIndex : USINT; (*0..3 = Array Requested*)
		IN_Scale : ARRAY[0..3] OF IN_Analog_Multiscale; (*0..3 = Arrays for Different Scale*)
	END_VAR
	VAR_OUTPUT
		OUT_Alarm : BOOL; (*Output Fault*)
		OUT_SpReached : BOOL; (*Output Set Point Reached*)
		OUT_RawOverflow : BOOL; (*Output Analog Fault*)
		OUT_RawUnderflow : BOOL; (*Output Analog Fault*)
		OUT_Scale : ARRAY[0..3] OF OUT_Analog_Multiscale;
	END_VAR
	VAR_IN_OUT
		IO : IO_Analog_IN_Type;
		HMI : HMI_Analog_Multiscale_Type;
	END_VAR
	VAR
		VAR_Fault : BOOL; (*Alarm Output for Fault or Warning*)
		VAR_Mask : BOOL;
		VAR_ChannelActive : BOOL;
		VAR_Wait : BOOL;
		VAR_iFault : BOOL;
		VAR_SpReached : BOOL;
		VAR_Index : USINT;
		VAR_Out : REAL;
		LCRLimScal_0_20mA : LCRLimScal;
		LCRLimScal_4_20mA : LCRLimScal;
		HMITotalizer : AnalogTotalizer;
		PLCCounter : AnalogTotalizer;
		TMR_TON_HighLimitDelay : TON;
		TMR_TON_LowLimitDelay : TON;
		TMR_TOF_SpReached : TOF;
	END_VAR
END_FUNCTION_BLOCK

FUNCTION_BLOCK Analog_In_Multicompare
	VAR_INPUT
		IN_ConfigPresent : BOOL;
		IN_Simulation : BOOL;
		IN_0_20mA : BOOL;
		IN_MaskEn : BOOL;
		IN_Reset : BOOL; (*Reset Analog Channel Alarm*)
		IN_FaultOutMode : USINT; (*LowOnFault(1) ; HighOnFault (2) HoldOnFault (0)*)
		IN_EngScale : BOOL;
		IN_AlarmEn : BOOL;
		IN_ConfigPopup : BOOL;
		IN_PLCCounterEn : BOOL;
		IN_CompareMode : USINT; (*0 = Off, 1 = PV_Greater_SP, 2 = PV_Less_SP, 3 = PV_Equal_SP, 4 = On*)
		IN_ScaleIndex : USINT; (*0..3 = Array Requested*)
		IN_Scale : ARRAY[0..3] OF IN_Analog_Multiscale; (*0..3 = Arrays for Different Scale*)
	END_VAR
	VAR_OUTPUT
		OUT_Alarm : BOOL; (*Output Fault*)
		OUT_SpReached : BOOL; (*Output Set Point Reached*)
		OUT_RawOverflow : BOOL; (*Output Analog Fault*)
		OUT_RawUnderflow : BOOL; (*Output Analog Fault*)
		OUT_Scale : ARRAY[0..3] OF OUT_Analog_Multiscale;
	END_VAR
	VAR_IN_OUT
		IO : IO_Analog_IN_Type;
		HMI : HMI_Analog_Multiscale_Type;
	END_VAR
	VAR
		VAR_Fault : BOOL; (*Alarm Output for Fault or Warning*)
		VAR_Mask : BOOL;
		VAR_ChannelActive : BOOL;
		VAR_Wait : BOOL;
		VAR_iFault : BOOL;
		VAR_SpReached : BOOL;
		VAR_Index : USINT;
		VAR_Out : REAL;
		LCRLimScal_0_20mA : LCRLimScal;
		LCRLimScal_4_20mA : LCRLimScal;
		HMITotalizer : AnalogTotalizer;
		PLCCounter : AnalogTotalizer;
		TMR_TON_HighLimitDelay : TON;
		TMR_TON_LowLimitDelay : TON;
		TMR_TOF_SpReached : TOF;
	END_VAR
END_FUNCTION_BLOCK

FUNCTION_BLOCK Digital_Obj
	VAR_INPUT
		IN_ConfigPresent : BOOL; (*Configuration: Device Present*)
		IN_Alarm : BOOL; (*Configuration: Timeout Alarm Control Enable*)
		IN_AlarmOnReq : BOOL; (*Control: On State Time Out Alarm Request*)
		IN_AlarmOffReq : BOOL; (*Control: Off State Time Out Alarm Request*)
		IN_SwitchDelay : TIME; (*Time: Row Input Switching State Display Delay*)
		IN_WaitOn : BOOL; (*Control: On State Wait Request*)
		IN_WaitOff : BOOL; (*Control: Off State Wait Request*)
		IN_OnDelay : TIME; (*Time: State On / Alarm On Time Delay*)
		IN_OffDelay : TIME; (*Time: State Off / Alarm Off Time Delay*)
		IN_Reset : BOOL; (*Control: Alarm Reset Push Button*)
		IN_MaskEn : BOOL; (*Control: Mask Enable*)
	END_VAR
	VAR_OUTPUT
		OUT : BOOL; (*State Switching Delayed*)
		OUT_OnDelayed : BOOL; (*State On Time Delayed*)
		OUT_OffDelayed : BOOL; (*State Off Time Delayed*)
		OUT_Alarm : BOOL; (*State On / Off Time Out Alarm*)
	END_VAR
	VAR_IN_OUT
		IO : IO_Digital_IN_Type; (*State: Digital Input Structure*)
		HMI : HMI_DI_Type;
	END_VAR
	VAR
		TMR_TON_SwOn : TON;
		TMR_TON_SwOff : TON;
		TMR_TON_OnTime : TON;
		TMR_TON_OffTime : TON;
		TMR_TON_OnAlarm : TON;
		TMR_TON_OffAlarm : TON;
		VAR_Signal : BOOL;
		VAR_Mask : BOOL;
	END_VAR
END_FUNCTION_BLOCK

FUNCTION_BLOCK Dosing_Obj (*//v1.7.4*)
	VAR_INPUT
		IN_Enable : BOOL; (*Enable*)
		IN_StartDosing : BOOL; (*Start dosing command*)
		IN_ChemicalPAA : BOOL; (*Type of chemical Acid PAA*)
		IN_ChemicalChlorine : BOOL; (*Type of chemical Chlorine*)
		IN_ChemicalOther : BOOL; (*Type of chemical Other*)
		IN_ChemicalDensity : REAL; (*Chemical density [kg/l]*)
		IN_FlowmeterPos : BOOL; (*Flowmeter position 0: Before dosing station 1: After dosing station*)
		IN_FlowmeterPulse : BOOL; (*Flowmeter pulse input*)
		IN_FlowmeterVolumePerPulse : REAL; (*Flowmeter volume per pulse [l]*)
		IN_VolumePerStroke : REAL; (*Chemical Solution volume dosed every pulse of the device [cm3]*)
		IN_ChemicalConcentration : REAL; (*Chemical Concentration [0..1000000 ppm]*)
		IN_ConcentrationSetPointRcp : REAL; (*Chemical Concentration Recipe Set-point [0..1000000 ppm] v1.7.4*)
		IN_DosingFBKCfg : BOOL; (*v1.7.4*)
		IN_DosingFBK : BOOL; (*Feedback from dosing device*)
		IN_TitrationCmd : BOOL; (*Titration comfirmation Command v1.7.5*)
		IN_ForceON : BOOL; (*Forced ON Command*)
		IN_ManualSetPointCondition : BOOL; (*Condition for manual SP v1.7.4*)
		IN_Clock : BOOL; (*Clock*)
	END_VAR
	VAR_OUTPUT
		OUT_DosingCMD : BOOL; (*Command to dosing device*)
	END_VAR
	VAR_IN_OUT
		HMI_DosingValues : HMI_DosingObj_Type; (*Chemical Concentration PV [0..1000000 ppm]*)
	END_VAR
	VAR
		VAR_OutCMD : BOOL;
		VAR_DosingCondition : BOOL;
		VAR_ChemicalDensity : REAL; (*Pure Chemical density [kg/l]*)
		VAR_SolutionDensity : REAL; (*Solution density [kg/l]*)
		VAR_DosingError : REAL; (*[l]*)
		VAR_RcipeConcentration : REAL; (*[%]*)
		VAR_WaterMassPerStroke : REAL; (*[kg]*)
		VAR_SolutionMassPerStroke : REAL; (*[kg]*)
		VAR_ChemicalMassPerStroke : REAL; (*[kg]*)
		VAR_WaterVolumePerStroke : REAL; (*[l]*)
		VAR_ChemicalVolumePerStroke : REAL; (*[l]*)
		VAR_TotalWater : REAL; (*[l]*)
		VAR_TotalChemical : REAL; (*[l]*)
		VAR_ActualConcentration : REAL; (*[0..1000000 ppm] v1.7.5*)
		VAR_ConcetrationSP : REAL; (*[0..1000000 ppm] v1.7.5*)
		VAR_TitrationDelta : REAL; (*[0..1000000 ppm] v1.7.5*)
		zzEdge00000 : BOOL;
		zzEdge00001 : BOOL;
		zzEdge00002 : BOOL;
		zzEdge00003 : BOOL;
		VAR_StrokeDone : BOOL; (*v1.7.4*)
		zzEdge00004 : BOOL;
	END_VAR
END_FUNCTION_BLOCK

FUNCTION_BLOCK Motor_Std_Fw_Bw
	VAR_INPUT
		IN_ConfigPresent : BOOL;
		IN_Simulation : BOOL;
		IN_Enable : BOOL; (*Safety OK ( True if not used)*)
		IN_AutoCnd : BOOL; (*Automation Logic Input*)
		IN_Backward : BOOL; (*Direction Reverse*)
		IN_Reset : BOOL; (*Fault Reset*)
		IN_HMIAutoForce : BOOL;
		IN_FbkCheck : BOOL;
		IN_ManEn : BOOL;
		IN_MaskEn : BOOL;
		IN_FBKDelay : TIME := T#500ms; (*Time: Running Control Delay*)
		IN_ConfigType : BOOL; (*Configuration: Type TRUE = Phoenix FALSE = Contactor*)
	END_VAR
	VAR_OUTPUT
		OUT_Running : BOOL; (*Motor On*)
		OUT_ContactorFBKFault : BOOL;
		OUT_OverloadFault : BOOL;
		OUT_Alarm : BOOL; (*Output for Alarm*)
		OUT_IsolatedFault : BOOL;
	END_VAR
	VAR_IN_OUT
		IO : IO_Motor_FwBw_Type;
		HMI : HMI_Motor_Type;
	END_VAR
	VAR
		TMR_TOF : TON;
		TMR_TON : TON;
		VAR_ContactorFBK : BOOL;
		VAR_DiFault : BOOL;
		VAR_Overload : BOOL;
		VAR_Mask : BOOL;
		VAR_Auto : BOOL;
		VAR_Fault : BOOL; (*Alarm Output for Fault or Warning*)
		VAR_FirstCycle : BOOL;
		VAR_Isolated : BOOL;
		zzEdge00000 : BOOL;
	END_VAR
END_FUNCTION_BLOCK

FUNCTION_BLOCK Motor_Std
	VAR_INPUT
		IN_ConfigPresent : BOOL;
		IN_Simulation : BOOL;
		IN_Enable : BOOL; (*Safety OK ( True if not used)*)
		IN_AutoCnd : BOOL; (*Automation Logic Input*)
		IN_Reset : BOOL; (*Fault Reset*)
		IN_HMIAutoForce : BOOL;
		IN_ManEn : BOOL;
		IN_MaskEn : BOOL;
		IN_FBKDelay : TIME := T#500ms; (*Time: Running Control Delay*)
		IN_ConfigType : BOOL; (*Configuration: Type TRUE = Phoenix FALSE = Contactor*)
	END_VAR
	VAR_OUTPUT
		OUT_Running : BOOL; (*Motor On*)
		OUT_IsolatedFault : BOOL;
		OUT_ContactorFBKFault : BOOL;
		OUT_OverloadFault : BOOL;
		OUT_Alarm : BOOL; (*Output for Alarm*)
	END_VAR
	VAR_IN_OUT
		IO : IO_Motor_Type;
		HMI : HMI_Motor_Type;
	END_VAR
	VAR
		TMR_TOF : TON;
		TMR_TON : TON;
		VAR_ContactorFBK : BOOL;
		VAR_Isolated : BOOL;
		VAR_Overload : BOOL;
		VAR_Mask : BOOL;
		VAR_Auto : BOOL;
		VAR_Fault : BOOL; (*Alarm Output for Fault or Warning*)
		VAR_FirstCycle : BOOL;
		zzEdge00000 : BOOL;
	END_VAR
END_FUNCTION_BLOCK

FUNCTION_BLOCK Motor_FC280_Vfd
	VAR_INPUT
		IN_Simulation : BOOL;
		IN_ConfigPresent : BOOL; (*Configuration: Device Present*)
		IN_Enable : BOOL;
		IN_AutoCnd : BOOL; (*Automation Logic Input*)
		IN_AutoSpeed : REAL;
		IN_Reverse : BOOL;
		IN_FrequencyMin : REAL;
		IN_FrequencyMax : REAL;
		IN_ManEn : BOOL; (*Control: Manual On Enabled*)
		IN_MaskEn : BOOL; (*Control: Alarm Mask Enable*)
		IN_Reset : BOOL; (*Control: Alarm Reset Push Button*)
		IN_HMIAutoForce : BOOL;
		IN_QuickStopCmd : BOOL; (*Control: Quick Stop Command (TRUE = Quick Stop)*)
		IN_JOGMode : BOOL; (*Control: JOG Mode (if TRUE)*)
		IN_JOGCnd : BOOL; (*Control: JOG Running Condition*)
		IN_CoastingCmd : BOOL; (*Control: Coasting (TRUE = Coasting)*)
		IN_FCD : BOOL; (*Configuration: Drive Type FCD V4.A.A.1.6.13*)
		IN_FBKDelay : TIME := T#500ms; (*Time: Running Control Delay*)
		IN_SafetyCtrlEn : BOOL; (*Configuration: Drive SafeOFF Enabled TRUE = Control Enabled*)
		IN_ScaleMax : REAL := 100.0; (*Configuration: Drive speed Scale Maximum Value*)
	END_VAR
	VAR_OUTPUT
		OUT_InOperation : BOOL;
		OUT_DriveSafetyFBKFault : BOOL; (*Safety XOR 37*)
		OUT_DriveFault : BOOL; (*Drive fault (from STW) or high current*)
		OUT_IsolatedFault : BOOL;
		OUT_OverloadFault : BOOL;
		OUT_ActualSpeed : REAL;
		OUT_ActualFrequency : REAL;
		OUT_ActualCurrent : REAL;
		OUT_ActualTorque : REAL;
		OUT_ActualPower : REAL;
		OUT_ActualSpeedRPM : REAL;
		OUT_Warning : BOOL; (*Drive warning (from STW)*)
		OUT_SpeedReferece : BOOL;
	END_VAR
	VAR_IN_OUT
		HMI_Danfoss : HMI_Danfoss_Diag_Type;
		HMI_Motor : HMI_Motor_FC_Type;
		IO_DanfossFC280 : IO_PLK_DanfossFC280_Drive_Type;
		IO_MotorFC280 : IO_MotorFC280_Type;
	END_VAR
	VAR
		VAR_RecSTW : Danfoss_STW_Type;
		VAR_RecDI : Danfoss_DI_Type; (*V4.A.A.1.6.13*)
		VAR_SendCTW : Danfoss_CTW_Type;
		TMR_TON_CurrentHigh : TON;
		TMR_TON_FaultFilter : TON;
		TMR_TON_FBKTimeOut : TON;
		TMR_TON_RFeedBack : TON;
		TMR_TON_WarningFilter : TON;
		VAR_CurrentHigh : BOOL;
		VAR_Event : Danfoss_Event_Type;
		VAR_Fault : BOOL; (*Memory Output Generic*)
		VAR_FirstCycle : BOOL;
		VAR_AutoSpeed : REAL;
		VAR_Isolated : BOOL;
		VAR_Overload : BOOL;
		VAR_Auto : BOOL;
		VAR_Mask : BOOL;
		VAR_Start : BOOL; (*Motor start*)
		zzEdge00000 : BOOL;
		zzEdge1 : BOOL;
	END_VAR
END_FUNCTION_BLOCK

FUNCTION_BLOCK Motor_Vfd
	VAR_INPUT
		IN_Simulation : BOOL;
		IN_ConfigPresent : BOOL; (*Configuration: Device Present*)
		IN_Enable : BOOL;
		IN_AutoCnd : BOOL; (*Automation Logic Input*)
		IN_AutoSpeed : REAL;
		IN_Reverse : BOOL;
		IN_FrequencyMin : REAL;
		IN_FrequencyMax : REAL;
		IN_ManEn : BOOL; (*Control: Manual On Enabled*)
		IN_MaskEn : BOOL; (*Control: Alarm Mask Enable*)
		IN_Reset : BOOL; (*Control: Alarm Reset Push Button*)
		IN_HMIAutoForce : BOOL;
		IN_QuickStopCmd : BOOL; (*Control: Quick Stop Command (TRUE = Quick Stop)*)
		IN_JOGMode : BOOL; (*Control: JOG Mode (if TRUE)*)
		IN_JOGCnd : BOOL; (*Control: JOG Running Condition*)
		IN_CoastingCmd : BOOL; (*Control: Coasting (TRUE = Coasting)*)
		IN_FCD : BOOL; (*Configuration: Drive Type FCD V4.A.A.1.6.13*)
		IN_FBKDelay : TIME := T#500ms; (*Time: Running Control Delay*)
		IN_SafetyCtrlEn : BOOL; (*Configuration: Drive SafeOFF Enabled TRUE = Control Enabled*)
		IN_ScaleMax : REAL := 100.0; (*Configuration: Drive speed Scale Maximum Value*)
	END_VAR
	VAR_OUTPUT
		OUT_InOperation : BOOL;
		OUT_DriveSafetyFBKFault : BOOL; (*Safety XOR 37*)
		OUT_DriveFault : BOOL; (*Drive fault (from STW) or high current*)
		OUT_IsolatedFault : BOOL;
		OUT_OverloadFault : BOOL;
		OUT_ActualSpeed : REAL;
		OUT_ActualFrequency : REAL;
		OUT_ActualCurrent : REAL;
		OUT_ActualTorque : REAL;
		OUT_ActualPower : REAL;
		OUT_ActualSpeedRPM : REAL;
		OUT_Warning : BOOL; (*Drive warning (from STW)*)
		OUT_SpeedReferece : BOOL;
		OUT_ActualDigitalState : Danfoss_DI_Type; (*V1.7.2*)
	END_VAR
	VAR_IN_OUT
		HMI_Danfoss : HMI_Danfoss_Diag_Type;
		HMI_Motor : HMI_Motor_FC_Type;
		IO_Danfoss : IO_PLK_Danfoss_Drive_Type;
		IO_Motor : IO_Motor_Type;
	END_VAR
	VAR
		VAR_RecSTW : Danfoss_STW_Type;
		VAR_RecDI : Danfoss_DI_Type; (*V4.A.A.1.6.13*)
		VAR_SendCTW : Danfoss_CTW_Type;
		TMR_TON_CurrentHigh : TON;
		TMR_TON_FaultFilter : TON;
		TMR_TON_FBKTimeOut : TON;
		TMR_TON_RFeedBack : TON;
		TMR_TON_WarningFilter : TON;
		VAR_CurrentHigh : BOOL;
		VAR_Event : Danfoss_Event_Type;
		VAR_Fault : BOOL; (*Memory Output Generic*)
		VAR_FirstCycle : BOOL;
		VAR_AutoSpeed : REAL;
		VAR_Isolated : BOOL;
		VAR_Overload : BOOL;
		VAR_Auto : BOOL;
		VAR_Mask : BOOL;
		VAR_Start : BOOL; (*Motor start*)
		zzEdge00000 : BOOL;
	END_VAR
END_FUNCTION_BLOCK

FUNCTION_BLOCK Valve_Dig_Mac (*Valve Control: Digital*)
	VAR_INPUT
		IN_ConfigPresent : BOOL; (*Configuration: Device Present*)
		IN_ConfigType : BOOL; (*Configuration: Device Type (0: Monostable - 1: Bistable)*)
		IN_Simulation : BOOL;
		IN_ConfigPositionSensorOpened : BOOL;
		IN_ConfigPositionSensorClosed : BOOL;
		IN_StrokeTime : TIME;
		IN_Enable : BOOL;
		IN_AutoCnd : BOOL; (*Automation Logic Input*)
		IN_EnableCnd : BOOL;
		IN_Cnd : BOOL;
		IN_FlipEnable : BOOL;
		IN_FlipRequest : BOOL;
		IN_FlipTime : TIME;
		IN_Reset : BOOL; (*Fault Reset*)
		IN_HMIAutoForce : BOOL;
		IN_ManEn : BOOL;
		IN_MaskEn : BOOL;
	END_VAR
	VAR_OUTPUT
		OUT : BOOL; (*Stroke done*)
		OUT_Alarm : BOOL; (*Fault Output for Alarm*)
		OUT_OpenedFiltered : BOOL; (*Stroke done*)
		OUT_ClosedFiltered : BOOL; (*Stroke done*)
		OUT_FlipDone : BOOL;
	END_VAR
	VAR_IN_OUT
		IO : IO_Valve_Type;
		HMI : HMI_Valve_Type;
	END_VAR
	VAR
		VAR_Enable : BOOL;
		VAR_iFault : BOOL;
		VAR_Mask : BOOL;
		TMR_TOF_FeedBackOpen : TOF;
		TMR_TOF_FeedBackClose : TOF;
		VAR_ManOn : BOOL;
		VAR_Auto : BOOL;
		MAX_Flip_Time : TIME := T#1S;
		VAR_AutoCnd : BOOL;
		VAR_ConfigPosition : BOOL;
		TMR_TON_ControlEnableDelay : TON;
		TMR_TON_Opened : TON;
		TMR_TON_Closed : TON;
		VAR_FeedBackOpen : BOOL;
		VAR_FeedBackClose : BOOL;
		VAR_ValveOpened : BOOL;
		VAR_Fault : BOOL;
		TMR_TP_Block : TP_Reset;
		TMR_TP_Release : TP_Reset;
		TMR_TON_Flip : TON;
		VAR_ValveClosed : BOOL;
		TMR_TON_ClosedFilter : TON;
		TMR_TON_OpenedFilter : TON;
	END_VAR
END_FUNCTION_BLOCK

FUNCTION_BLOCK Valve_Dig (*Valve Control: Digital*)
	VAR_INPUT
		IN_ConfigPresent : BOOL; (*Configuration: Device Present*)
		IN_ConfigType : BOOL; (*Configuration: Device Type (0: Monostable - 1: Bistable)*)
		IN_ConfigNormallyOpen : BOOL; (*Configuration: Device Type (0: Normally Closed - 1: Normally Open) v1.5*)
		IN_Simulation : BOOL;
		IN_ConfigPositionSensorOpened : BOOL;
		IN_ConfigPositionSensorClosed : BOOL;
		IN_StrokeTime : TIME;
		IN_Enable : BOOL;
		IN_AutoCnd : BOOL; (*Automation Logic Input*)
		IN_EnableCnd : BOOL;
		IN_Cnd : BOOL;
		IN_FlipEnable : BOOL;
		IN_FlipRequest : BOOL;
		IN_FlipTime : TIME;
		IN_Reset : BOOL; (*Fault Reset*)
		IN_HMIAutoForce : BOOL;
		IN_ManEn : BOOL;
		IN_MaskEn : BOOL;
	END_VAR
	VAR_OUTPUT
		OUT : BOOL; (*Stroke done*)
		OUT_Alarm : BOOL; (*Fault Output for Alarm*)
		OUT_OpenedFiltered : BOOL; (*Stroke done*)
		OUT_ClosedFiltered : BOOL; (*Stroke done*)
		OUT_FlipDone : BOOL;
	END_VAR
	VAR_IN_OUT
		IO : IO_Valve_Type;
		HMI : HMI_Valve_Type;
	END_VAR
	VAR
		VAR_Enable : BOOL;
		VAR_iFault : BOOL;
		VAR_Mask : BOOL;
		TMR_TOF_FeedBackOpen : TOF;
		TMR_TOF_FeedBackClose : TOF;
		VAR_ManOn : BOOL;
		VAR_Auto : BOOL;
		MAX_Flip_Time : TIME := T#1S;
		VAR_AutoCnd : BOOL;
		VAR_ConfigPosition : BOOL;
		TMR_TON_ControlEnableDelay : TON;
		TMR_TON_Opened : TON;
		TMR_TON_Closed : TON;
		VAR_FeedBackOpen : BOOL;
		VAR_FeedBackClose : BOOL;
		VAR_ValveOpened : BOOL;
		VAR_Fault : BOOL;
		TMR_TON_Flip : TON;
		VAR_ValveClosed : BOOL;
		TMR_TON_ClosedFilter : TON;
		TMR_TON_OpenedFilter : TON;
	END_VAR
END_FUNCTION_BLOCK

FUNCTION_BLOCK Valve_Mod
	VAR_INPUT
		IN_ConfigPresent : BOOL;
		IN_Simulation : BOOL;
		IN_ConfigPositionSensorOpened : BOOL;
		IN_ConfigPositionSensorClosed : BOOL;
		IN_ConfigPositionAnalogFBK : BOOL;
		IN_StrokeTime : TIME;
		IN_ConfigNormallyOpen : BOOL;
		IN_Enable : BOOL;
		IN_AutoCnd : BOOL;
		IN_AutoVal : REAL;
		IN_OpeningRampEn : BOOL;
		IN_OpeningRampValue : REAL;
		IN_ClosingRampEn : BOOL;
		IN_ClosingRampValue : REAL;
		IN_OutMin : REAL; (*Min Opening [%]*)
		IN_OutMax : REAL; (*Max Opening [%]*)
		IN_HMIAutoForce : BOOL;
		IN_ManEn : BOOL;
		IN_MaskEn : BOOL;
		IN_Reset : BOOL; (*Fault Reset*)
	END_VAR
	VAR_OUTPUT
		OUT_Cv : REAL; (*Analog output (0.0 - 100.0)*)
		OUT_Alarm : BOOL; (*Falt Output for Alarm*)
		OUT_RampDone : BOOL; (*Ramp Done*)
		OUT_FBKFault : BOOL;
		OUT_FBK : REAL; (*Analog Input FeedBack Value 0.0 - 100.0%*)
	END_VAR
	VAR_IN_OUT
		IO : IO_Valve_Mod_Type;
		HMI : HMI_Valve_Mod_Type;
	END_VAR
	VAR
		VAR_Fault : BOOL; (*Falt Output for Alarm*)
		VAR_iFault : BOOL;
		VAR_ConfigPosition : BOOL;
		VAR_OutMan : REAL;
		VAR_Open : REAL;
		VAR_iOpen : REAL;
		TMR_TOF_DOValveOn : TOF;
		VAR_FirstCycle : BOOL;
		VAR_DOValveOn : BOOL;
		VAR_DOValveOff : BOOL;
		VAR_DIFeedBackOpen : BOOL;
		VAR_DIFeedBackClose : BOOL;
		VAR_Mask : BOOL;
		TMR_TON_PositionFiltered : TON;
		VAR_ManOn : BOOL;
		VAR_Auto : BOOL;
		LCRMovingRamp : LCRRamp;
		VAR_OpeningRamp : REAL;
		VAR_ClosingRamp : REAL;
		LCRLimScal_AO : LCRLimScal;
		LCRLimScal_AI : LCRLimScal;
		VAR_FaultSensorOn : BOOL;
		VAR_FaultSensorOff : BOOL;
		VAR_FaultSensorFBK : BOOL;
	END_VAR
END_FUNCTION_BLOCK

FUNCTION_BLOCK Fan_Obj
	VAR_INPUT
		IN_ConfigPresent : BOOL;
		IN_RoofType : BOOL; (*0: Fan 1: Galvani*)
		IN_GalvaniRoofFlowSet : BOOL;
		IN_CgfHmiLampOn : BOOL;
		IN_FanNumber : USINT := 1;
		IN_AutoSpeed : REAL;
		IN_Enable : BOOL;
		IN_HMIAutoForce : BOOL;
		IN_Reset : BOOL; (*Control: Alarm Reset Push Button*)
	END_VAR
	VAR_OUTPUT
		OUT_Alarm : BOOL;
		Out_Light : BOOL; (*v4.A.A.1.7.0*)
		OUT_OverloadFault : BOOL;
	END_VAR
	VAR_IN_OUT
		IO : IO_FanMain_Type;
		HMI : HMI_Fan_Type;
		ALARM : FanZoneAlarm_Type;
	END_VAR
	VAR
		TMR_TON_OnDelay : ARRAY[1..6] OF TON;
		TMR_TON_OffDelay : ARRAY[1..6] OF TON;
		VAR_Auto : ARRAY[1..6] OF BOOL;
		TMR_TON_OnDelay_Gal : TON;
		TMR_TON_OffDelay_Gal : TON;
		VAR_Auto_Gal : BOOL;
		VAR_OUT : REAL;
		VAR_GalvaniOn : BOOL;
		VAR_GalvaniFlowSet : BOOL;
		VAR_AbsoluteFilter : BOOL;
		VAR_Overload : BOOL; (*//v1.7.4*)
		VAR_PreFilter : BOOL;
		VAR_RunFeedback : BOOL; (*//v1.7.4*)
		VAR_ResetHMI : BOOL;
		VAR_i : USINT;
	END_VAR
END_FUNCTION_BLOCK

FUNCTION_BLOCK MotionFan_Obj
	VAR_INPUT
		IN_ConfigPresent : BOOL;
		IN_Enable : BOOL; (*Safety OK ( True if not used)*)
		IN_AutoCnd : BOOL; (*Automation Logic Input*)
		IN_Reset : BOOL; (*Fault Reset*)
		IN_FBKDelay : TIME := T#500ms; (*Time: Running Control Delay*)
	END_VAR
	VAR_OUTPUT
		OUT_Running : BOOL; (*Motor On*)
		OUT_IsolatedFault : BOOL;
		OUT_ContactorFBKFault : BOOL;
		OUT_OverloadFault : BOOL;
		OUT_Alarm : BOOL; (*Output for Alarm*)
	END_VAR
	VAR_IN_OUT
		IO : IO_MotionFan_Type;
	END_VAR
	VAR
		TMR_TOF : TON;
		TMR_TON : TON;
		VAR_ContactorFBK : BOOL;
		VAR_Isolated : BOOL;
		VAR_Overload : BOOL;
		VAR_Fault : BOOL; (*Alarm Output for Fault or Warning*)
	END_VAR
END_FUNCTION_BLOCK
(*Shift Register Object*)

FUNCTION_BLOCK CapPhotoCell_SftObj_old (* *) (*$GROUP=User,$CAT=User,$GROUPICON=User.png,$CATICON=User.png*)
	VAR_INPUT
		IN_ConfigPresent : BOOL; (*Configuration: Device Present*)
		IN_Enable : BOOL; (*Configuration: Enable *)
		IN_Alarm : BOOL; (*Configuration: Timeout Alarm Control Enable*)
		IN_WaitOn : BOOL; (*Control: On State Wait Request*)
		IN_WaitOff : BOOL; (*Control: Off State Wait Request*)
		IN_MachinePitch : BOOL; (*Control: Machine Pitch Pulse*)
		IN_ResetCounters : BOOL;
		IN_MaskEn : BOOL; (*Control: Mask Enable*)
		IN_GrippersNumber : USINT; (*Control : Grip Number For Repetitive Control*)
		IN_CBlockAbsoluteValue : USINT; (*Control: Container Stop Threshold For Absolute Container Lack*)
		IN_CBlockRepetitiveValue : USINT; (*Control: Container Stop Threshold For Repetitive Container Lack*)
		IN_MStopAbsoluteValue : USINT; (*Control: Critical Stop Threshold For Absolute Container Lack*)
		IN_MStopConsecutiveValue : USINT; (*Control: Critical Stop Threshold For Consecutive Container Lack*)
	END_VAR
	VAR_OUTPUT
		OUT : BOOL; (*State Switching Delayed*)
		OUT_CBlockRepetitive : BOOL; (*Container Stop For Repetitive Lack Errors*)
		OUT_CBlockAbsolute : BOOL; (*Container Stop For Absolute Lack Errors*)
		OUT_MStopConsecutive : BOOL; (*Critical Stop For Consecutive*)
		OUT_MStopAbsolute : BOOL; (*Critical Stop For Absolute*)
		OUT_AlwaysTrueError : BOOL;
	END_VAR
	VAR_IN_OUT
		IO : IO_Digital_IN_Type; (*State: Digital Input Structure*)
		HMI : HMI_Photocell_Type;
		SHIFT_Position : UINT;
	END_VAR
	VAR CONSTANT
		CST_AlwaysTrueMaxSteps : USINT := 10; (*Max Number Of Steps With The Photocell Always TRUE*)
		CST_RepetitiveArrayDim : USINT := 50; (*Repetitive Array Dimension*)
	END_VAR
	VAR
		TMR_TON_TotalCounterReset : TON;
		VAR_Mask : BOOL;
		VAR_Signal : BOOL;
		VAR_CounterResetMemory : BOOL;
		VAR_TotalCounterResetMemory : BOOL;
		VAR_EdgeChecked : BOOL;
		VAR_GrippersNumber : USINT;
		VAR_ActualValveCounter : USINT := 1;
		VAR_RepetitiveCounterArray : ARRAY[1..CST_RepetitiveArrayDim] OF USINT;
	END_VAR
END_FUNCTION_BLOCK

FUNCTION_BLOCK CapPhotoCell_SftObj (* *) (*$GROUP=User,$CAT=User,$GROUPICON=User.png,$CATICON=User.png*)
	VAR_INPUT
		IN_ConfigPresent : BOOL; (*Configuration: Device Present*)
		IN_Enable : BOOL; (*Configuration: Enable *)
		IN_Alarm : BOOL; (*Configuration: Timeout Alarm Control Enable*)
		IN_WaitOn : BOOL; (*Control: On State Wait Request*)
		IN_WaitOff : BOOL; (*Control: Off State Wait Request*)
		IN_MachinePitch : BOOL; (*Control: Machine Pitch Pulse*)
		IN_ResetCounters : BOOL; (*V1.61 Reset Absolute Errors*)
		IN_ResetCountersConsecutive : BOOL; (*V1.61 Reset Consecutive errors*)
		IN_MaskEn : BOOL; (*Control: Mask Enable*)
		IN_GrippersNumber : USINT; (*Control : Grip Number For Repetitive Control*)
		IN_CBlockAbsoluteValue : USINT; (*Control: Container Stop Threshold For Absolute Container Lack*)
		IN_CBlockAbsoluteQuantity : UINT; (*Control: Critical Stop Threshold For Consecutive Container Lack*)
		IN_CBlockRepetitiveValue : USINT; (*Control: Container Stop Threshold For Repetitive Container Lack*)
		IN_MStopConsecutiveValue : USINT; (*Control: Critical Stop Threshold For Consecutive Container Lack*)
	END_VAR
	VAR_OUTPUT
		OUT : BOOL; (*State Switching Delayed*)
		OUT_CBlockRepetitive : BOOL; (*Container Stop For Repetitive Lack Errors*)
		OUT_CBlockAbsolute : BOOL; (*Container Stop For Absolute Lack Errors*)
		OUT_MStopConsecutive : BOOL; (*Critical Stop For Consecutive*)
		OUT_AlwaysTrueError : BOOL;
	END_VAR
	VAR_IN_OUT
		IO : IO_Digital_IN_Type; (*State: Digital Input Structure*)
		HMI : HMI_Photocell_Type;
		SHIFT_Position : UINT;
	END_VAR
	VAR CONSTANT
		CST_AlwaysTrueMaxSteps : USINT := 10; (*Max Number Of Steps With The Photocell Always TRUE*)
		CST_CounterArrayDim : USINT := 50; (*Repetitive Array Dimension*)
	END_VAR
	VAR
		TMR_TON_TotalCounterReset : TON;
		VAR_AbsoluteErrorN : USINT := 1;
		VAR_Mask : BOOL;
		VAR_Signal : BOOL;
		VAR_CounterResetMemory : BOOL;
		VAR_CounterConsResetMemory : BOOL; (*V1.61*)
		VAR_TotalCounterResetMemory : BOOL;
		VAR_EdgeChecked : BOOL;
		VAR_GrippersNumber : USINT;
		VAR_ActualValveCounter : USINT := 1;
		VAR_i : USINT;
		VAR_CapsReleased : UDINT;
		VAR_AbsoluteCounterArray : ARRAY[1..CST_CounterArrayDim] OF UDINT;
		VAR_RepetitiveCounterArray : ARRAY[1..CST_CounterArrayDim] OF USINT;
	END_VAR
END_FUNCTION_BLOCK

FUNCTION_BLOCK Ejector_SftObj (* Container Ejector Valve *)
	VAR_INPUT
		IN_ConfigPresent : BOOL; (*Configuration: Device Present*)
		IN_ConfigType : BOOL; (*Configuration: Device Type (0: Monostable - 1: Bistable)*)
		IN_Enable : BOOL;
		IN_MachinePitch : BOOL;
		IN_FillingErrorEject : BOOL;
		IN_SamplingModeActive : BOOL; (*V1.61*)
		IN_ResetCounters : BOOL;
		IN_HMIAutoForce : BOOL;
		IN_ManEn : BOOL;
		IN_MaskEn : BOOL;
		IN_ShiftPosition : UINT;
		IN_CBlockAbsoluteValue : USINT; (*Control: Container Stop Threshold For Absolute Container Lack*)
		IN_MStopConsecutiveValue : USINT; (*Control: Machine Stop Threshold For Consecutive Container Lack*)
	END_VAR
	VAR_OUTPUT
		OUT : BOOL; (*Stroke done*)
		OUT_CBlockAbsolute : BOOL; (*Container Stop For Absolute Lack Errors*)
		OUT_MStopConsecutive : BOOL; (*Critical Stop For Consecutive*)
	END_VAR
	VAR_IN_OUT
		IO : IO_Valve_Type;
		HMI : HMI_Valve_Ejector_Type;
	END_VAR
	VAR
		TMR_TON_TotalCounterReset : TON;
		VAR_Mask : BOOL;
		VAR_ManOn : BOOL;
		VAR_Auto : BOOL;
		VAR_AutoCnd : BOOL;
		VAR_CounterResetMemory : BOOL;
		VAR_TotalCounterResetMemory : BOOL;
		VAR_ValveOpened : BOOL;
		VAR_ValveClosed : BOOL;
	END_VAR
END_FUNCTION_BLOCK

FUNCTION_BLOCK PhotoCell_SftObj (* *) (*$GROUP=User,$CAT=User,$GROUPICON=User.png,$CATICON=User.png*)
	VAR_INPUT
		IN_ConfigPresent : BOOL; (*Configuration: Device Present*)
		IN_Enable : BOOL; (*Configuration: Enable *)
		IN_Alarm : BOOL; (*Configuration: Alarm Control Enable*)
		IN_WaitOn : BOOL; (*Control: On State Wait Request*)
		IN_WaitOff : BOOL; (*Control: Off State Wait Request*)
		IN_MachinePitch : BOOL; (*Control: Machine Pitch Pulse*)
		IN_ResetCounters : BOOL;
		IN_WritePresenceEnable : BOOL; (*Configuration Type of Photocell (0: Disabel Write Presence, 1: Enable Write Presence)*)
		IN_MaskEn : BOOL; (*Control: Mask Enable*)
		IN_GrippersNumber : USINT; (*Control : Grip Number For Repetitive Control*)
		IN_CBlockAbsoluteValue : USINT; (*Control: Container Stop Threshold For Absolute Container Lack*)
		IN_CBlockRepetitiveValue : USINT; (*Control: Container Stop Threshold For Repetitive Container Lack*)
		IN_MStopAbsoluteValue : USINT; (*Control: Machine Stop Threshold For Absolute Container Lack*)
		IN_MStopConsecutiveValue : USINT; (*Control: Machine Stop Threshold For Consecutive Container Lack*)
	END_VAR
	VAR_OUTPUT
		OUT : BOOL; (*State Switching Delayed*)
		OUT_CBlockRepetitive : BOOL; (*Container Stop For Repetitive Lack Errors*)
		OUT_CBlockAbsolute : BOOL; (*Container Stop For Absolute Lack Errors*)
		OUT_MStopConsecutive : BOOL; (*Critical Stop For Consecutive*)
		OUT_MStopAbsolute : BOOL; (*Critical Stop For Absolute*)
		OUT_AlwaysTrueError : BOOL;
	END_VAR
	VAR_IN_OUT
		IO : IO_Digital_IN_Type; (*State: Digital Input Structure*)
		HMI : HMI_Photocell_Type;
		SHIFT_Position : UINT;
	END_VAR
	VAR CONSTANT
		CST_AlwaysTrueMaxSteps : USINT := 10; (*Max Number Of Steps With The Photocell Always TRUE*)
		CST_RepetitiveArrayDim : USINT := 50; (*Repetitive Array Dimension*)
	END_VAR
	VAR
		TMR_TON_TotalCounterReset : TON;
		VAR_Mask : BOOL;
		VAR_Signal : BOOL;
		VAR_CounterResetMemory : BOOL;
		VAR_TotalCounterResetMemory : BOOL;
		VAR_EdgeChecked : BOOL;
		VAR_GrippersNumber : USINT;
		VAR_ActualValveCounter : USINT := 1;
		VAR_RepetitiveCounterArray : ARRAY[1..CST_RepetitiveArrayDim] OF USINT;
	END_VAR
END_FUNCTION_BLOCK
```

#### HMI_Structure.typ
```iecst
(*VALVES*)

TYPE
	HMI_Valve_Type : 	STRUCT  (*Valves Structure: Digital*)
		Out : BOOL; (*State: Output*)
		Alarm : BOOL; (*State: Position Alarm *)
		Opened : BOOL; (*State: Feed-Back Opened*)
		Closed : BOOL; (*State: Feed-Back Closed*)
		ConfigPosition : BOOL; (*Configuration: Valve Feed-Back Position Present *)
		ConfigPresent : BOOL; (*Configuration: Device Present*)
		ManOff : BOOL; (*Command: Manual Closed*)
		ManOn : BOOL; (*Command: Manual Opened *)
		Mask : BOOL; (*Command: Position Alarm Mask*)
		ManEnable : BOOL; (*Command Enable: Manual Enabled*)
		MaskEnable : BOOL; (*Command Enable: Mask Enabled*)
	END_STRUCT;
	HMI_Valve_MixProof_Type : 	STRUCT  (*Valves Structure: Digital Mix Proof*)
		Out : BOOL; (*State: Output*)
		Alarm : BOOL; (*State: Position Alarm *)
		Opened : BOOL; (*State: Feed-Back Opened*)
		Closed : BOOL; (*State: Feed-Back Closed*)
		ConfigPosition : BOOL; (*Configuration: Valve Feed-Back Position Present *)
		ConfigPresent : BOOL; (*Configuration: Device Present*)
		ManOff : BOOL; (*Command: Manual Closed*)
		ManOn : BOOL; (*Command: Manual Opened *)
		Mask : BOOL; (*Command: Position Alarm Mask*)
		ManEnable : BOOL; (*Command Enable: Manual Enabled*)
		MaskEnable : BOOL; (*Command Enable: Mask Enabled*)
		H_Out : BOOL; (*High State: Output*)
		H_Alarm : BOOL; (*High State: Position Alarm *)
		H_Opened : BOOL; (*High State: Feed-Back Opened*)
		H_Closed : BOOL; (*High State: Feed-Back Closed*)
		H_ConfigPosition : BOOL; (*High Configuration: Valve Closed State Present *)
		H_ManOff : BOOL; (*High Command: Manual Closed*)
		H_ManOn : BOOL; (*High Command: Manual Opened *)
		H_Mask : BOOL; (*High Command: Position Alarm Mask*)
		H_ManEnable : BOOL; (*High Command Enable: Manual Enabled*)
		H_MaskEnable : BOOL; (*High Command Enable: Mask Enabled*)
		L_Out : BOOL; (*Low State: Output*)
		L_Alarm : BOOL; (*Low State: Position Alarm *)
		L_Opened : BOOL; (*Low State: Feed-Back Opened*)
		L_Closed : BOOL; (*Low State: Feed-Back Closed*)
		L_ConfigPosition : BOOL; (*Low Configuration: Valve Closed State Present *)
		L_ManOff : BOOL; (*Low Command: Manual Closed*)
		L_ManOn : BOOL; (*Low Command: Manual Opened *)
		L_Mask : BOOL; (*Low Command: Position Alarm Mask*)
		L_ManEnable : BOOL; (*Low Command Enable: Manual Enabled*)
		L_MaskEnable : BOOL; (*Low Command Enable: Mask Enabled*)
	END_STRUCT;
	HMI_Valve_Mod_Type : 	STRUCT  (*Valves Structure: Analogic*)
		Out : BOOL; (*State: Output*)
		Alarm : BOOL; (*State: Position Alarm *)
		Opened : BOOL; (*State: Feed-Back Opened*)
		Closed : BOOL; (*State: Feed-Back Closed*)
		ConfigSlew : BOOL; (*Configuration: Output Slew Present*)
		ConfigPosition : BOOL; (*Configuration: Valve Feed-Back Position Present *)
		ConfigPresent : BOOL; (*Configuration: Device Present*)
		ManOff : BOOL; (*Command: Manual Closed*)
		ManOn : BOOL; (*Command: Drive Manual OUT = OUT_Man*)
		Mask : BOOL; (*Command: Position Alarm Mask*)
		ManEnable : BOOL; (*Command Enable: Manual Enabled*)
		MaskEnable : BOOL; (*Command Enable: Mask Enabled*)
		OUT_CV : REAL; (*State: Actual OUTPUT Control Value (0.0-:-100.0)*)
		OUT_Man : REAL; (*Command: Manual OUTPUT Value (0.0-:-100.0)*)
		FBK : REAL; (*State: Feed-Back INPUT Value (0.0-:-100.0)*)
	END_STRUCT;
END_TYPE

(*MOTORS*)

TYPE
	HMI_SCU_Type : 	STRUCT
		Visibility : BOOL;
		Alarm : BOOL;
		ErrCode : DINT;
		HwCmdUp : BOOL;
		HwCmdDown : BOOL;
		HwCmdStorePosition : BOOL;
	END_STRUCT;
	HMI_Column_Type : 	STRUCT
		Visibility : BOOL;
		Running : BOOL; (*State: Output*)
		Current : REAL;
		Initialized : BOOL;
		Position : REAL;
		Alarm : BOOL;
	END_STRUCT;
	HMI_Motor_Type : 	STRUCT  (*Motor Structure: Direct On Line*)
		Out : BOOL; (*State: Running*)
		Alarm : BOOL; (*State: Alarm (Isolated, Overload, FBK Fault)*)
		Isolated : BOOL; (*State: Motor Isolated*)
		Overload : BOOL; (*State: Overload*)
		FeedBack : BOOL; (*State: Feed-Back Fault*)
		ConfigPresent : BOOL; (*Configuration: Device Present*)
		ManOff : BOOL; (*Command: Manual Stop*)
		ManOn : BOOL; (*Command: Manual Start*)
		Mask : BOOL; (*Command: Alarm Mask*)
		ManEnable : BOOL; (*Command Enable: Manual Enabled*)
		MaskEnable : BOOL; (*Command Enable: Mask Enabled*)
	END_STRUCT;
	HMI_Motor_FC_Type : 	STRUCT  (*Motor Structure: Variable Frequency Drive*)
		Out : BOOL; (*State: Running *)
		Alarm : BOOL; (*State: Alarm (Isolated, Overload, FBK Fault)*)
		Isolated : BOOL; (*State: Motor Isolated*)
		Overload : BOOL; (*State: Overload*)
		FeedBack : BOOL; (*State: In Operation/Safe-OFF Feed-Back Fault*)
		BusFault : BOOL; (*State: Bus Control Fault*)
		Fault : BOOL; (*State: Inverter Internal Fault*)
		ConfigPresent : BOOL; (*Configuration: Device Present*)
		ManOff : BOOL; (*Command: Manual Stop*)
		ManOn : BOOL; (*Command: Manual Start*)
		Mask : BOOL; (*Command: Alarm Mask*)
		ManEnable : BOOL; (*Command Enable: Manual Enabled*)
		MaskEnable : BOOL; (*Command Enable: Mask Enabled*)
		OUT_CV : REAL; (*State: Actual OUTPUT Value (0.0-:-100.0)*)
		OUT_Man : REAL; (*Command: Manual OUTPUT Value (0.0-:-100.0)*)
	END_STRUCT;
	HMI_Dosing_Pump_Type : 	STRUCT  (*Motor Structure: Dosing Pump*)
		Out : BOOL; (*State: Running *)
		Alarm : BOOL; (*State: Alarm (Isolated, Overload, FBK Fault)*)
		Isolated : BOOL; (*State: Motor Isolated*)
		Overload : BOOL; (*State: Overload*)
		FeedBack : BOOL; (*State: In Operation/Safe-OFF Feed-Back Fault*)
		Pulse_FBK : BOOL; (*State: Pulse Feed-Back Alarm*)
		Internal_Fault : BOOL; (*State: Internal Alarm*)
		ConfigPresent : BOOL; (*Configuration: Device Present*)
		ManOff : BOOL; (*Command: Manual Stop*)
		ManOn : BOOL; (*Command: Manual Start *)
		Mask : BOOL; (*Command: Alarm Mask*)
		ManEnable : BOOL; (*Command Enable: Manual Enabled*)
		MaskEnable : BOOL; (*Command Enable: Mask Enabled*)
		Stroke_Value : REAL; (*Setting CC/Stroke [cm3/stroke]*)
		Concentration : REAL; (*Tank Concentrated percentage [0..1000000 ppm]*)
		Density : REAL; (*Specific Weight [kg]*)
	END_STRUCT;
	HMI_Danfoss_Diag_Type : 	STRUCT
		PCV : HMI_Danfoss_PCV_Type;
		PCD_Read : HMI_Danfoss_PCD_Read_Type;
	END_STRUCT;
	HMI_Danfoss_PCV_Type : 	STRUCT
		Alarm : DINT;
	END_STRUCT;
	HMI_Danfoss_PCD_Read_Type : 	STRUCT
		Power : REAL;
		Motor_Current : REAL;
		Frequency : REAL;
		Torque : REAL;
		Main_Actual_Value : REAL;
		Speed_RPM : REAL;
		Status_Word : UINT;
	END_STRUCT;
	HMI_Fan_Type : 	STRUCT
		HMI_Pressurizer : ARRAY[1..6]OF HMI_Pressurizer_Type; (*Single Fans to HMI*)
		HMI_Galvani : HMI_Galvani_Type; (*Galvani Roof Fans*)
	END_STRUCT;
	HMI_Galvani_Type : 	STRUCT
		Out : BOOL;
		ConfigPresent : BOOL; (*Configuration: Device Present*)
		SS2P_Lamp1 : HMI_SS2P_Type; (*SS2P Lamp*)
		SS2P_Lamp2 : HMI_SS2P_Type; (*SS2P Lamp*)
		ManState : BOOL; (*State: Device in manual mode*)
		ManEnable : BOOL; (*Command Enable: Manual Enabled*)
		ManFlowSet : BOOL; (*Command: Manual Flow set command*)
		ManOff : BOOL; (*Command: Manual Stop*)
		ManOn : BOOL; (*Command: Manual Start*)
		MaskEnable : BOOL; (*Command Enable: Mask Enabled*)
		Mask : BOOL; (*Command: Alarm Mask*)
		FlowSet : BOOL; (*State: Flow set speed *)
		Alarm : BOOL; (*State: Alarm (Isolated, Overload, FBK Fault)*)
		AlarmAbsoluteFilter : BOOL; (*Fault : Absolute filter clogged*)
		AlarmPrefilterExt : BOOL; (*Fault : External PreFilter Clogged*)
		AlarmPrefilterInt : BOOL; (*Fault : Internal PreFilter Clogged*)
		Overload : BOOL; (*State: Power supply on*)
	END_STRUCT;
	HMI_Pressurizer_Type : 	STRUCT
		Out : BOOL;
		ConfigPresent : BOOL; (*Configuration: Device Present*)
		SS2P_Lamp : HMI_SS2P_Type; (*SS2P Lamp*)
		ManState : BOOL; (*State: Device in manual mode*)
		ManEnable : BOOL; (*Command Enable: Manual Enabled*)
		ManOff : BOOL; (*Command: Manual Stop*)
		ManOn : BOOL; (*Command: Manual Start*)
		MaskEnable : BOOL; (*Command Enable: Mask Enabled*)
		Mask : BOOL; (*Command: Alarm Mask*)
		OUT_Man : REAL; (*Command :  Manual Speed OUT value selected (0 - 100)*)
		OUT_CV : REAL; (*State : Actual Speed OUT value %*)
		Alarm : BOOL; (*State: Alarm (Isolated, Overload, FBK Fault)*)
		AlarmFilter : BOOL; (*Fault : Absolute filter or PreFilter Clogged*)
	END_STRUCT;
	HMI_GreasingPump_Type : 	STRUCT
		LowLevel : HMI_DI_Type;
		CycleEnd : HMI_DI_Type;
		Motor : HMI_Motor_Type;
	END_STRUCT;
END_TYPE

(*INSTRUMENTS*)

TYPE
	HMI_Valve_Ejector_Type : 	STRUCT  (*Valves Structure: Digital*)
		Out : BOOL; (*State: Output*)
		Alarm : BOOL; (*State: Position Alarm *)
		Opened : BOOL; (*State: Feed-Back Opened*)
		Closed : BOOL; (*State: Feed-Back Closed*)
		ConfigPosition : BOOL; (*Configuration: Valve Feed-Back Position Present *)
		ConfigPresent : BOOL; (*Configuration: Device Present*)
		ManOff : BOOL; (*Command: Manual Closed*)
		ManOn : BOOL; (*Command: Manual Opened *)
		Mask : BOOL; (*Command: Position Alarm Mask*)
		ManEnable : BOOL; (*Command Enable: Manual Enabled*)
		MaskEnable : BOOL; (*Command Enable: Mask Enabled*)
		CounterReset : BOOL; (*Command: Reset Counter*)
		TotalErrors : UDINT; (*State : Total Errors*)
		AbsoluteErrors : USINT; (*State : Absolute Errors*)
		ConsecutiveErrors : USINT; (*State : Consecutive Errors*)
	END_STRUCT;
	HMI_Photocell_Type : 	STRUCT  (*Instrument Structure: Photocell*)
		On : BOOL; (*State: Active*)
		Alarm : BOOL; (*State: Alarm*)
		Wait : BOOL; (*State: Waiting condition*)
		ConfigAlarm : BOOL; (*Configuration: Alarm Present*)
		ConfigPresent : BOOL; (*Configuration: Instrument Present*)
		Mask : BOOL; (*Command: Alarm Mask*)
		MaskEnable : BOOL; (*Command Enable: Mask Enabled*)
		CounterReset : BOOL; (*Command: Reset Counter*)
		TotalErrors : UDINT; (*State : Total Errors*)
		RepetitiveErrors : USINT; (*State : Repetitive Errors*)
		AbsoluteErrors : USINT; (*State : Absolute Errors*)
		ConsecutiveErrors : USINT; (*State : Consecutive Errors*)
		AlwaysTrueSteps : USINT;
	END_STRUCT;
	HMI_DI_Type : 	STRUCT  (*Instrument Structure: Digital*)
		On : BOOL; (*State: Active*)
		Alarm : BOOL; (*State: Alarm*)
		Wait : BOOL; (*State: Waiting condition*)
		ConfigAlarm : BOOL; (*Configuration: Alarm Present*)
		ConfigPresent : BOOL; (*Configuration: Instrument Present*)
		Mask : BOOL; (*Command: Alarm Mask*)
		MaskEnable : BOOL; (*Command Enable: Mask Enabled*)
	END_STRUCT;
	HMI_Analog_IN_Type : 	STRUCT  (*Instrument Structure: Analogic*)
		Alarm : BOOL; (*State: Instrument in fault (Probe Fault)*)
		Wait : BOOL; (*State: Waiting condition*)
		WaitCounter : BOOL; (*State: Waiting Counter condition*)
		ConfigPopUp : BOOL; (*Configuration: Instrument Pop-Up Present (TRUE=Pop-Up NOT Present)*)
		ConfigTot : BOOL; (*Configuration: Totalizator Present (TRUE=Totalizator Present)*)
		ConfigAlarm : BOOL; (*Configuration: Alarm Present (TRUE=Command Mask Present)*)
		ConfigPresent : BOOL; (*Configuration: Instrument Present*)
		ConfigCounter : BOOL; (*Configuration: Counter Present*)
		ResetTot : BOOL; (*Command: Totalizator Reset*)
		Mask : BOOL; (*Command: Alarm Mask (Probe Fault disabled)*)
		MaskEnable : BOOL; (*Command Enable: Mask Enabled*)
		PV : REAL; (*Input: Scaled Process Value*)
		SP : REAL; (*Input: Actual SetPoint*)
		PV_Counter : REAL; (*Input: Counter Current Value*)
		SP_Counter : REAL; (*Input: Counter Requested Value*)
		Tot : REAL; (*Input: Totalizator*)
	END_STRUCT;
	HMI_Analog_IN_Mode_Type : 	STRUCT  (*Instrument Structure: Analogic Multi Scale*)
		Mode : ARRAY[0..3]OF HMI_Analog_IN_Type;
	END_STRUCT;
	HMI_Analog_Multiscale_Type : 	STRUCT  (*Instrument Structure: Analogic*)
		Alarm : BOOL; (*State: Instrument in fault (Probe Fault)*)
		Unit : USINT; (*0 = Unit1 ; 1 = Unit2 ; 2 = Unit3 ; etc...*)
		ConfigPopup : BOOL; (*Configuration: Instrument Pop-Up Present (TRUE=Pop-Up NOT Present)*)
		ConfigAlarm : BOOL; (*Configuration: Alarm Present (TRUE=Command Mask Present)*)
		ConfigPresent : BOOL; (*Configuration: Instrument Present*)
		ResetTot : BOOL; (*Command: Totalizator Reset*)
		Mask : BOOL; (*Command: Alarm Mask (Probe Fault disabled)*)
		MaskEnable : BOOL; (*Command Enable: Mask Enabled*)
		Wait : ARRAY[0..3]OF BOOL; (*State: Waiting condition*)
		ConfigTot : ARRAY[0..3]OF BOOL; (*Configuration: Totalizator Present (TRUE=Totalizator Present)*)
		WaitCounter : ARRAY[0..3]OF BOOL; (*State: Waiting Counter condition*)
		ConfigCounter : ARRAY[0..3]OF BOOL; (*Configuration: Counter Present*)
		PV : ARRAY[0..3]OF REAL; (*Input: Scaled Process Value*)
		SP : ARRAY[0..3]OF REAL; (*Input: Actual SetPoint*)
		PV_Counter : ARRAY[0..3]OF REAL; (*Input: Counter Current Value*)
		SP_Counter : ARRAY[0..3]OF REAL; (*Input: Counter Requested Value*)
		Tot : ARRAY[0..3]OF REAL; (*Input: Totalizator*)
	END_STRUCT;
	HMI_TNK_Level_Type : 	STRUCT
		CFG_Level_Percentage : BOOL;
		Level_Percentage : REAL; (*[%]*)
		CFG_Level_Percentage_SP : BOOL; (*[%]*)
		Level_Height_SP : REAL; (*[mm]*)
		Level_Percentage_SP : REAL; (*[%]*)
		CFG_Volume : BOOL;
		Volume : REAL; (*[l]*)
		CFG_Volume_SP : BOOL; (*[l]*)
		Level_Percentage_Wait : BOOL;
		Level_Height_Wait : BOOL;
		Volume_Wait : BOOL;
		Volume_SP : REAL; (*[l]*)
		CFG_Level_Height : BOOL;
		Level_Height : REAL; (*[mm]*)
	END_STRUCT;
	HMI_TNK_Level_v00_Type : 	STRUCT
		ConfigPresent : BOOL := TRUE;
		TNK_Height_mm : REAL; (*[mm]*)
		TNK_Height_Sp : REAL; (*[mm]*)
		TNK_Height_Wait : BOOL;
		TNK_Percentage : REAL; (*[%]*)
		TNK_Percentage_Sp : REAL; (*[%]*)
		TNK_Percentage_Wait : BOOL;
		TNK_Volume_liters : REAL; (*[l]*)
		TNK_Volume_Sp : REAL; (*[l]*)
		TNK_Volume_Wait : BOOL;
	END_STRUCT;
	HMI_GateDoor_Type : 	STRUCT
		Opened : BOOL;
		ShortSafety : BOOL;
		Production : HMI_DI_Type;
		Cleaning : HMI_DI_Type;
	END_STRUCT;
END_TYPE

(*PID*)

TYPE
	HMI_PID_Mode_Type : 	STRUCT
		Mode : ARRAY[0..3]OF HMI_PID_Type;
	END_STRUCT;
	HMI_PID_Type : 	STRUCT  (*PID Structure: PID Control*)
		Enable : BOOL; (*State: PID Enable*)
		Mode : BOOL; (*State: PID Mode (Automatic = 1  Manual = 0)*)
		Alarm : BOOL; (*State: PID PV in fault*)
		SP_Obtained : BOOL; (*State: PID Set Point Reached*)
		SP_SlewRunning : BOOL; (*State: PID Set Point Slew Running*)
		CnScale : BOOL; (*Configuration: FF and PID OUT Scale - TRUE-> 0-100%, FALSE-> Ing.Unit.*)
		ConfigSlewPresent : BOOL; (*Configuration: Slew Present*)
		ConfigPresent : BOOL; (*Configuration : PID present*)
		SPLocal : BOOL; (*Command: PID Manual Set Point -> "SP_Local"*)
		PV : REAL; (*State: PID Process Value*)
		SP_Actual : REAL; (*State: PID Set Point in Use*)
		SP_Target : REAL; (*State: PID Set Point*)
		FF_OUT : REAL; (*State: PID Feed Forward calculated value*)
		OUT : REAL; (*State: PID Output*)
		SP_Local : REAL; (*Command: PID Manual Set Point Target Value*)
	END_STRUCT;
END_TYPE

(*PWM*)

TYPE
	HMI_PWM_Type : 	STRUCT  (*PWM Structure: Pulse Width Modulation*)
		Out : BOOL; (*State: On*)
		Alarm : BOOL; (*State: Alarm (Isolated, Overload, FBK Fault)*)
		Isolated : BOOL; (*State: Isolated*)
		Overload : BOOL; (*State: Overload*)
		FeedBack : BOOL; (*State: Feed-Back Fault*)
		ConfigPresent : BOOL; (*Configuration: Device Present*)
		ManOff : BOOL; (*Command: Manual Stop*)
		ManOn : BOOL; (*Command: Manual Start*)
		Mask : BOOL; (*Command: Alarm Mask*)
		ManEnable : BOOL; (*Command Enable: Manual Enabled*)
		MaskEnable : BOOL; (*Command Enable: Mask Enabled*)
		OUT_CV : REAL; (*State: Actual OUTPUT Control Value (0.0-:-100.0)*)
		OUT_Man : REAL; (*Command: Manual OUTPUT Value (0.0-:-100.0)*)
	END_STRUCT;
END_TYPE

(*SS2P*)

TYPE
	HMI_SS2P_Type : 	STRUCT  (*Selector 2 position (Auto-Man; ON-OFF;) 0=Auto/OFF - 1=Man/ON*)
		Enable : BOOL; (*State: Command Enabled*)
		LampON : BOOL; (*State: Lamp Command ON*)
		Blink : BOOL; (*State: Blink LampOn*)
		Visibility : BOOL; (*Configuration: Present*)
		ON : BOOL; (*Command: Selector Button ON*)
	END_STRUCT;
END_TYPE

(*DOSING*)

TYPE
	HMI_DosingObj_Type : 	STRUCT
		Total_Water : REAL;
		Total_Chemical : REAL;
		Actual_Concentration : REAL;
		Actual_SetPoint : REAL; (*v1.7.4*)
		Manual_SetPoint : REAL; (*v1.7.4*)
		Titration_Value_Act : REAL; (*v1.7.5*)
		Titration_Value_Old : REAL; (*v1.7.5*)
		Titration_Time_Preset : UINT; (*v1.7.5*)
		Titration_Time_Actual : UINT; (*v1.7.5*)
	END_STRUCT;
END_TYPE
```

#### IO_Structure.typ
```iecst
(*VALVES*)

TYPE
	IO_Valve_Mod_Type : 	STRUCT
		AO_Raw : INT;
		AI_Raw : INT;
		Valve : IO_Valve_Type;
	END_STRUCT;
	IO_Valve_Type : 	STRUCT
		DI_Opened : BOOL; (*DI Valve Open - Feedback*)
		DI_Closed : BOOL; (*DI Valve Close - Feedback*)
		DO_Opened : BOOL; (*DO Valve Open*)
		DO_Closed : BOOL; (*DO Valve Close*)
	END_STRUCT;
END_TYPE

(*MOTORS*)

TYPE
	IO_Motor_FwBw_Type : 	STRUCT  (*Motor control Forward Backward*)
		DI_SafetyEnable : BOOL; (*Safety Enable from IOMapping*)
		DI_SafetyFault : BOOL; (*Safety Feed-Back from Safety CPU*)
		DI_Fault : BOOL;
		DI_ContactorFBK : BOOL; (*Contactor Feed-Back *)
		DI_OverloadOK : BOOL := TRUE; (*Not present in case of UL*)
		DI_ManSwitchON : BOOL := TRUE;
		DO_MotorFw : BOOL; (*Start Forward*)
		DO_MotorBw : BOOL; (*Start Backward*)
	END_STRUCT;
	IO_MotorFC280_Type : 	STRUCT  (*Motor control*)
		DI_SafetyEnable : BOOL; (*Safety Enable from IOMapping*)
		DI_SafetyFault : BOOL; (*Safety Feed-Back from Safety CPU*)
		DI_ManSwitchON : BOOL := TRUE;
		DI_ContactorFBK : BOOL; (*Contactor Feed-Back *)
		DI_OverloadOK : BOOL := TRUE; (*Not present in case of UL*)
		DO_MotorON : BOOL; (*Start*)
		DO_ShuntTrip : BOOL; (*Thermal Protection Forced Trip*)
	END_STRUCT;
	IO_Motor_Type : 	STRUCT  (*Motor control*)
		DI_SafetyEnable : BOOL; (*Safety Enable from IOMapping*)
		DI_SafetyFault : BOOL; (*Safety Feed-Back from Safety CPU*)
		DI_ManSwitchON : BOOL := TRUE;
		DI_ContactorFBK : BOOL; (*Contactor Feed-Back *)
		DI_OverloadOK : BOOL := TRUE; (*Not present in case of UL*)
		DO_MotorON : BOOL; (*Start*)
		DO_ShuntTrip : BOOL; (*Thermal Protection Forced Trip*)
	END_STRUCT;
	IO_PLK_DanfossFC280_Drive_Type : 	STRUCT  (*Powerlink Danfoss VLT Interface*)
		Input : IO_PLK_DanfossFC280_IN;
		Output : IO_PLK_DanfossFC280_OUT;
	END_STRUCT;
	IO_PLK_Danfoss_Drive_Type : 	STRUCT  (*Powerlink Danfoss VLT Interface*)
		Input : IO_PLK_Danfoss_IN;
		Output : IO_PLK_Danfoss_OUT;
	END_STRUCT;
	IO_PLK_DanfossFC280_IN : 	STRUCT  (*Powerlink Danfoss VLT Inputs*)
		STW : UINT; (*Status Word*)
		MAV : INT; (*Main Actual Value*)
		ActFreq : UDINT; (*Actual Frequency [Hz]*)
		ActCurrent : UINT; (*Actual Current [A]*)
		Power : UDINT; (*Power [kW]*)
		Torque : DINT; (*Torque [Nm]*)
		SpeedRPM : DINT; (*Speed [RPM]*)
		STW_EX : UDINT; (*Extended Status Word 1*)
		ErrorCode : UDINT; (*Error Code 1*)
		DigitalInput : UINT; (*Digital Input V4.A.A.1.6.13*)
	END_STRUCT;
	IO_PLK_Danfoss_IN : 	STRUCT  (*Powerlink Danfoss VLT Inputs*)
		STW : UINT; (*Status Word*)
		MAV : INT; (*Main Actual Value*)
		ActFreq : UINT; (*Actual Frequency [Hz]*)
		ActCurrent : DINT; (*Actual Current [A]*)
		Power : DINT; (*Power [kW]*)
		Torque : INT; (*Torque [Nm]*)
		SpeedRPM : DINT; (*Speed [RPM]*)
		STW_EX : UDINT; (*Extended Status Word 1*)
		ErrorCode : UDINT; (*Error Code 1*)
		DigitalInput : UINT; (*Digital Input V4.A.A.1.6.13*)
	END_STRUCT;
	IO_PLK_DanfossFC280_OUT : 	STRUCT  (*Powerlink Danfoss VLT Outputs*)
		CTW : UINT; (*Control Word*)
		MRW : INT; (*Main Reference Value*)
	END_STRUCT;
	IO_PLK_Danfoss_OUT : 	STRUCT  (*Powerlink Danfoss VLT Outputs*)
		CTW : UINT; (*Control Word*)
		MRW : INT; (*Main Reference Value*)
	END_STRUCT;
	IO_FanMain_Type : 	STRUCT
		DI_OverloadOK : BOOL := TRUE;
		DO_ZoneLighting : BOOL; (*V4.A.A.1.7.0*)
		Pressurizer : ARRAY[1..6]OF IO_Pressurizer_Type;
		GalvaniRoof : IO_GalvaniRoof_Type;
	END_STRUCT;
	IO_PressurizerMain_Type : 	STRUCT
		DI_OverloadOK : BOOL := TRUE;
		Pressurizer : ARRAY[1..6]OF IO_Pressurizer_Type;
	END_STRUCT;
	IO_GalvaniRoof_Type : 	STRUCT
		DI_Running : BOOL;
		DI_AbsoluteFilterAlarm : BOOL;
		DI_PrefilterExtAlarm : BOOL;
		DI_PrefilterIntAlarm : BOOL;
		DI_CabinetPoweredOn : BOOL;
		DO_Start : BOOL;
		DO_FlowSet : BOOL;
		DO_LightingArea_1 : BOOL;
		DO_LightingArea_2 : BOOL;
	END_STRUCT;
	IO_Pressurizer_Type : 	STRUCT
		DO_Lighting : BOOL;
		AO_Raw : INT;
		DI_PressurizerON : BOOL; (*Pressurizzer ON*)
		DI_PrefilterAlarm : BOOL; (*Pressurizzer prefilter clogged*)
		DI_AbsoluteFilterAlarm : BOOL; (*Pressurizzer absolute filter clogged*)
		DI_OverloadOK : BOOL := TRUE; (*//v1.7.4*)
	END_STRUCT;
	IO_MotionFan_Type : 	STRUCT
		DI_ManSwitchON : BOOL := TRUE;
		DI_OverloadOK : BOOL := TRUE;
		DI_ContactorFBK : BOOL := TRUE;
		DO_MotorON : BOOL;
	END_STRUCT;
END_TYPE

(*INSTRUMENTS*)

TYPE
	IO_Analog_IN_OUT_Type : 	STRUCT
		AO_Raw : INT := 0; (*Analog Input From HW*)
		AI : IO_Analog_IN_Type; (*Analog Input From HW*)
	END_STRUCT;
	IO_Analog_IN_Type : 	STRUCT
		AI_Raw : INT := 0; (*Analog Input From HW*)
		DI_ChannelOk : BOOL := TRUE;
		DI_Pulse : BOOL; (*Totalizer Pulse*)
		DI_Alarm : BOOL; (*Instrument Alarm*)
		DO_SetScale : BOOL; (*Scale Change Output*)
	END_STRUCT;
	IO_Digital_IN_Type : 	STRUCT
		DI_Input : BOOL;
	END_STRUCT;
	IO_Digital_OUT_Type : 	STRUCT
		DO_Output : BOOL;
	END_STRUCT;
	IO_GreasingPump_Type : 	STRUCT
		LowLevel : IO_Digital_IN_Type;
		CycleEnd : IO_Digital_IN_Type;
		Motor : IO_Motor_Type;
	END_STRUCT;
	IN_Analog_Multiscale : 	STRUCT
		ScaleLOW : REAL;
		ScaleHIGH : REAL;
		ActualSP : REAL; (*Signal Input Actual Set Point*)
		MinDev : REAL; (*To Set Point Low Deviation (for SP obtained)*)
		MaxDev : REAL; (*To Set Point High Deviation (for SP obtained)*)
		WaitDelay : TIME;
		HighLimitEn : BOOL;
		HighLimitSP : REAL;
		HighLimitHyst : REAL;
		HighLimitDelay : TIME;
		LowLimitEn : BOOL;
		LowLimitSP : REAL;
		LowLimitHyst : REAL;
		LowLimitDelay : TIME;
		TotPulseWeight : REAL;
		TotType : USINT;
		PLCCounterSP : REAL;
		PLCCounterReset : BOOL;
		HMITotEn : BOOL;
		HMITotReset : BOOL;
	END_STRUCT;
	OUT_Analog_Multiscale : 	STRUCT
		ActValue : REAL; (*Manipulated value*)
		LowLimit : BOOL;
		HighLimit : BOOL;
		PLCCounterReached : BOOL; (*Output Fault*)
		Active : BOOL; (*Request to Instrument Scale Activation*)
	END_STRUCT;
	IO_IncrementalEncoder : 	STRUCT  (*//V4.A.A.1.6.11*)
		CountAtZero : DINT;
		Counter : INT;
		Status : USINT;
		Reference : USINT;
		DI_EnableReference : IO_Digital_IN_Type;
		DI_NotPowered : IO_Digital_IN_Type;
	END_STRUCT;
END_TYPE
```
